(* IEC 61131-3 sources: std_i2980_v2.06_cp053/Source/IMM/ieccontrol/ODC1 (part 10) *)

@BEG_Export

@BEG_Algo
@POSTUPDATE_ALGORITHM @RT(21)pProgramSwitchChanged @STRUCTURED_TEXT
@RT(0) @RT(24)sv_bProgramSwitchChanged @RT(9)PU_Task_3 @F @F
@END_Algo

@BEG_Dcl
@RT(16)DclTreeContainer
0
@END_Dcl

@END_Export

@BEG_Export

@BEG_Algo
@POSTUPDATE_ALGORITHM @RT(18)pActivationChanged @STRUCTURED_TEXT
@RT(0) @RT(21)sv_bActivationChanged @RT(9)PU_Task_3 @F @F
@END_Algo

@BEG_Dcl
@RT(16)DclTreeContainer
0
@END_Dcl

@END_Export

@BEG_Export

@BEG_Algo
@PROCESS_ALGORITHM @RT(13)paVersionInfo @STRUCTURED_TEXT
@RT(0) @RT(0) @RT(8)TaskSlow @T @F
@END_Algo

@BEG_Dcl
@RT(16)DclTreeContainer
1
@Var @RT(1)b @RT(0) @T @F @DT @RT(4)BOOL @RT(0) @T @T @BASIC 0 @F
@F @F
@T
@BEG_Attrib
3 @RT(0) @RT(0) @RT(0)
@END_Attrib
1 0 @F @F @F @F

@END_Dcl

@END_Export

@BEG_Export

@BEG_Algo
@POSTUPDATE_ALGORITHM @RT(24)pChangeToProgramSwitches @STRUCTURED_TEXT
@RT(0) @RT(22)sv_bUseProgramSwitches @RT(9)PU_Task_7 @F @F
@END_Algo

@BEG_Dcl
@RT(16)DclTreeContainer
1
@Var @RT(7)iDevice @RT(0) @T @F @DT @RT(4)DINT @RT(0) @T @T @BASIC 0 @F
@F @F
@T
@BEG_Attrib
3 @RT(0) @RT(0) @RT(0)
@END_Attrib
1 4 @F @F @F @F

@END_Dcl

@END_Export

@BEG_Export

@BEG_Algo
@ALGORITHM @RT(26)aCheckCycleStartConditions @STRUCTURED_TEXT
@RT(0) @RT(0) @RT(0) @F @F
@END_Algo

@BEG_Dcl
@RT(16)DclTreeContainer
10
@Var @RT(3)Pos @RT(0) @T @T @DERIVED 0 @T @T @DT @RT(12)tsODCStepPos @RT(0) @T @T @UNKNOWN 0 @F
@F @F
@T
@BEG_Attrib
3 @RT(0) @RT(0) @RT(0)
@END_Attrib
1 0 @F @F @F @F

@Var @RT(8)DeviceId @RT(0) @T @T @DERIVED 0 @T @T @DT @RT(10)tsDeviceId @RT(0) @T @T @UNKNOWN 0 @F
@F @F
@T
@BEG_Attrib
3 @RT(0) @RT(0) @RT(0)
@END_Attrib
1 0 @F @F @F @F

@Var @RT(11)SafetyArray @RT(0) @T @T @DERIVED 0 @T @T @DT @RT(20)tyODCDependencyArray @RT(0) @T @T @UNKNOWN 0 @F
@F @F
@T
@BEG_Attrib
3 @RT(0) @RT(0) @RT(0)
@END_Attrib
1 0 @F @F @F @F

@Var @RT(12)iDefaultMove @RT(0) @T @F @DT @RT(4)DINT @RT(0) @T @T @BASIC 0 @F
@F @F
@T
@BEG_Attrib
3 @RT(0) @RT(0) @RT(0)
@END_Attrib
1 0 @F @F @F @F

@Var @RT(7)iDevice @RT(0) @T @F @DT @RT(4)DINT @RT(0) @T @T @BASIC 0 @F
@F @F
@T
@BEG_Attrib
3 @RT(0) @RT(0) @RT(0)
@END_Attrib
1 4 @F @F @F @F

@Var @RT(8)bAllowed @RT(0) @T @F @DT @RT(4)BOOL @RT(0) @T @T @BASIC 0 @F
@F @F
@T
@BEG_Attrib
3 @RT(0) @RT(0) @RT(0)
@END_Attrib
1 0 @F @F @F @F

@Var @RT(22)abODCCheckDependencies @RT(0) @T @T @DERIVED 0 @T @T @DT @RT(22)ABODCCheckDependencies @RT(0) @T @T @UNKNOWN 0 @F
@F @F
@T
@BEG_Attrib
3 @RT(0) @RT(0) @RT(0)
@END_Attrib
1 0 @F @F @F @F

@Var @RT(17)fbCheckPosReached @RT(0) @T @T @DERIVED 0 @T @T @DT @RT(17)FBCheckPosReached @RT(0) @T @T @UNKNOWN 0 @F
@F @F
@T
@BEG_Attrib
3 @RT(0) @RT(0) @RT(0)
@END_Attrib
1 0 @F @F @F @F

@Var @RT(15)bEjectorIgnored @RT(0) @T @F @DT @RT(4)BOOL @RT(0) @T @T @BASIC 0 @F
@F @F
@T
@BEG_Attrib
3 @RT(0) @RT(0) @RT(0)
@END_Attrib
1 0 @F @F @F @F

@Var @RT(17)EjectorDependency @RT(0) @T @F @DT @RT(5)LWORD @RT(0) @T @T @BASIC 0 @F
@F @F
@T
@BEG_Attrib
3 @RT(0) @RT(0) @RT(0)
@END_Attrib
1 0 @F @F @F @F

@END_Dcl

@END_Export

@BEG_Export

@BEG_Algo
@POSTUPDATE_ALGORITHM @RT(14)pOperationMode @STRUCTURED_TEXT
@RT(0) @RT(16)sv_OperationMode @RT(9)PU_Task_7 @F @F
@END_Algo

@BEG_Dcl
@RT(16)DclTreeContainer
2
@Var @RT(10)PrevOpMode @RT(0) @T @T @DERIVED 0 @T @T @DT @RT(15)tnOperationMode @RT(0) @T @T @UNKNOWN 0 @F
@F @F
@T
@BEG_Attrib
3 @RT(7)nManual @RT(0) @RT(0)
@END_Attrib
1 0 @F @F @F @F

@Var @RT(14)sOperationMode @RT(0) @T @F @DT @RT(11)STRING(255) @RT(0) @T @T @STRING 0 @F @RT(3)255 @F
@F @F
@T
@BEG_Attrib
3 @RT(0) @RT(0) @RT(0)
@END_Attrib
1 4 @F @F @F @F

@END_Dcl

@END_Export

@BEG_Export

@BEG_Algo
@PROCESS_ALGORITHM @RT(27)paRunManualCombinedMovement @SEQUENTIAL_FLOW_CHART
@RT(0) @RT(0) @RT(13)TaskSequencer @F @F
@END_Algo

@BEG_Dcl
@RT(16)DclTreeContainer
0
@END_Dcl

@END_Export

@BEG_Export

@BEG_Algo
@PROCESS_ALGORITHM @RT(23)paCheckConditionsManual @STRUCTURED_TEXT
@RT(0) @RT(0) @RT(10)TaskAnalog @F @F
@END_Algo

@BEG_Dcl
@RT(16)DclTreeContainer
2
@Var @RT(10)TmpStepPos @RT(0) @T @T @DERIVED 0 @T @T @DT @RT(12)tsODCStepPos @RT(0) @T @T @UNKNOWN 0 @F
@F @F
@T
@BEG_Attrib
3 @RT(0) @RT(0) @RT(0)
@END_Attrib
1 0 @F @F @F @F

@Var @RT(1)i @RT(0) @T @F @DT @RT(4)DINT @RT(0) @T @T @BASIC 0 @F
@F @F
@T
@BEG_Attrib
3 @RT(0) @RT(0) @RT(0)
@END_Attrib
1 4 @F @F @F @F

@END_Dcl

@END_Export

@BEG_Export

@BEG_Algo
@PROCESS_ALGORITHM @RT(11)paCycleTime @STRUCTURED_TEXT
@RT(0) @RT(0) @RT(10)TaskInject @F @F
@END_Algo

@BEG_Dcl
@RT(16)DclTreeContainer
2
@Var @RT(1)b @RT(0) @T @F @DT @RT(4)BOOL @RT(0) @T @T @BASIC 0 @F
@F @F
@T
@BEG_Attrib
3 @RT(0) @RT(0) @RT(0)
@END_Attrib
1 0 @F @F @F @F

@Var @RT(14)fbTonCycleTime @RT(0) @T @T @DERIVED 0 @T @T @DT @RT(3)TON @RT(0) @T @T @UNKNOWN 0 @F
@F @F
@T
@BEG_Attrib
3 @RT(0) @RT(0) @RT(0)
@END_Attrib
1 0 @F @F @F @F

@END_Dcl

@END_Export

@BEG_Export

@BEG_Algo
@PROCESS_ALGORITHM @RT(18)paCycleTimeMachine @STRUCTURED_TEXT
@RT(0) @RT(0) @RT(7)TaskMid @F @F
@END_Algo

@BEG_Dcl
@RT(16)DclTreeContainer
2
@Var @RT(1)b @RT(0) @T @F @DT @RT(4)BOOL @RT(0) @T @T @BASIC 0 @F
@F @F
@T
@BEG_Attrib
3 @RT(0) @RT(0) @RT(0)
@END_Attrib
1 0 @F @F @F @F

@Var @RT(21)fbTonCycleTimeMachine @RT(0) @T @T @DERIVED 0 @T @T @DT @RT(3)TON @RT(0) @T @T @UNKNOWN 0 @F
@F @F
@T
@BEG_Attrib
3 @RT(0) @RT(46)Clock the cycletime from start to end of cycle @RT(0)
@END_Attrib
1 0 @F @F @F @F

@END_Dcl

@END_Export

@BEG_Export

@BEG_Algo
@POSTUPDATE_ALGORITHM @RT(21)pSequenceInterruption @STRUCTURED_TEXT
@RT(0) @RT(24)sv_bSequenceInterruption @RT(10)PU_Task_13 @F @F
@END_Algo

@BEG_Dcl
@RT(16)DclTreeContainer
1
@Var @RT(5)dummy @RT(0) @T @F @DT @RT(4)DINT @RT(0) @T @T @BASIC 0 @F
@F @F
@T
@BEG_Attrib
3 @RT(0) @RT(0) @RT(0)
@END_Attrib
1 0 @F @F @F @F

@END_Dcl

@END_Export

@BEG_Export

@BEG_Algo
@ALGORITHM @RT(21)aStartInverseMovement @STRUCTURED_TEXT
@RT(0) @RT(0) @RT(0) @F @F
@END_Algo

@BEG_Dcl
@RT(16)DclTreeContainer
5
@Var @RT(7)iMoveNr @RT(0) @T @F @DT @RT(4)DINT @RT(0) @T @T @BASIC 0 @F
@F @F
@T
@BEG_Attrib
3 @RT(0) @RT(0) @RT(0)
@END_Attrib
1 1 @F @F @F @F

@Var @RT(7)iColumn @RT(0) @T @F @DT @RT(4)DINT @RT(0) @T @T @BASIC 0 @F
@F @F
@T
@BEG_Attrib
3 @RT(0) @RT(0) @RT(0)
@END_Attrib
1 1 @F @F @F @F

@Var @RT(8)iFuIndex @RT(0) @T @F @DT @RT(4)DINT @RT(0) @T @T @BASIC 0 @F
@F @F
@T
@BEG_Attrib
3 @RT(0) @RT(0) @RT(0)
@END_Attrib
1 0 @F @F @F @F

@Var @RT(14)iMoveIdInverse @RT(0) @T @T @DERIVED 0 @T @T @DT @RT(10)tMoveIdent @RT(0) @T @T @UNKNOWN 0 @F
@F @F
@T
@BEG_Attrib
3 @RT(0) @RT(0) @RT(0)
@END_Attrib
1 0 @F @F @F @F

@Var @RT(1)i @RT(0) @T @F @DT @RT(4)DINT @RT(0) @T @T @BASIC 0 @F
@F @F
@T
@BEG_Attrib
3 @RT(0) @RT(0) @RT(0)
@END_Attrib
1 4 @F @F @F @F

@END_Dcl

@END_Export

@BEG_Export

@BEG_Algo
@POSTUPDATE_ALGORITHM @RT(8)pStepFwd @STRUCTURED_TEXT
@RT(0) @RT(10)di_StepFwd @RT(9)PU_Task_3 @F @F
@END_Algo

@BEG_Dcl
@RT(16)DclTreeContainer
0
@END_Dcl

@END_Export

@BEG_Export

@BEG_Algo
@POSTUPDATE_ALGORITHM @RT(8)pStepBwd @STRUCTURED_TEXT
@RT(0) @RT(10)di_StepBwd @RT(9)PU_Task_3 @F @F
@END_Algo

@BEG_Dcl
@RT(16)DclTreeContainer
2
@Var @RT(7)iColumn @RT(0) @T @F @DT @RT(4)DINT @RT(0) @T @T @BASIC 0 @F
@F @F
@T
@BEG_Attrib
3 @RT(0) @RT(0) @RT(0)
@END_Attrib
1 4 @F @F @F @F

@Var @RT(13)iActiveMoveNr @RT(0) @T @F @DT @RT(4)DINT @RT(0) @T @T @BASIC 0 @F
@F @F
@T
@BEG_Attrib
3 @RT(0) @RT(0) @RT(0)
@END_Attrib
1 0 @F @F @F @F

@END_Dcl

@END_Export

@BEG_Export

@BEG_Algo
@EVENT_ALGORITHM @RT(28)evaModifyCycleStartCondition @STRUCTURED_TEXT
@RT(0) @RT(27)evModifyCycleStartCondition @RT(9)EV_Task_3 @F @F
@END_Algo

@BEG_Dcl
@RT(16)DclTreeContainer
8
@Var @RT(26)evModifyCycleStartCondData @RT(0) @T @T @DERIVED 0 @T @T @DT @RT(27)tevModifyCycleStartCondData @RT(0) @T @T @UNKNOWN 0 @F
@F @F
@T
@BEG_Attrib
3 @RT(0) @RT(0) @RT(0)
@END_Attrib
1 1 @F @F @F @F

@Var @RT(5)dummy @RT(0) @T @F @DT @RT(4)DINT @RT(0) @T @T @BASIC 0 @F
@F @F
@T
@BEG_Attrib
3 @RT(0) @RT(0) @RT(0)
@END_Attrib
1 0 @F @F @F @F

@Var @RT(9)eventData @RT(0) @T @T @DERIVED 0 @T @T @DT @RT(27)tevModifyCycleStartCondData @RT(0) @T @T @UNKNOWN 0 @F
@F @F
@T
@BEG_Attrib
3 @RT(0) @RT(0) @RT(0)
@END_Attrib
1 0 @F @F @F @F

@Var @RT(8)iFuIndex @RT(0) @T @F @DT @RT(4)DINT @RT(0) @T @T @BASIC 0 @F
@F @F
@T
@BEG_Attrib
3 @RT(0) @RT(0) @RT(0)
@END_Attrib
1 0 @F @F @F @F

@Var @RT(1)i @RT(0) @T @F @DT @RT(4)DINT @RT(0) @T @T @BASIC 0 @F
@F @F
@T
@BEG_Attrib
3 @RT(0) @RT(0) @RT(0)
@END_Attrib
1 4 @F @F @F @F

@Var @RT(7)iMoveNr @RT(0) @T @F @DT @RT(4)DINT @RT(0) @T @T @BASIC 0 @F
@F @F
@T
@BEG_Attrib
3 @RT(0) @RT(0) @RT(0)
@END_Attrib
1 0 @F @F @F @F

@Var @RT(15)fbAddDependency @RT(0) @T @T @DERIVED 0 @T @T @DT @RT(15)FBAddDependency @RT(0) @T @T @UNKNOWN 0 @F
@F @F
@T
@BEG_Attrib
3 @RT(0) @RT(0) @RT(0)
@END_Attrib
1 0 @F @F @F @F

@Var @RT(15)fbGetMoveNumber @RT(0) @T @T @DERIVED 0 @T @T @DT @RT(15)FBGetMoveNumber @RT(0) @T @T @UNKNOWN 0 @F
@F @F
@T
@BEG_Attrib
3 @RT(0) @RT(0) @RT(0)
@END_Attrib
1 0 @F @F @F @F

@END_Dcl

@END_Export

@BEG_Body
@TL(14)
(**************************************** WARNING ********************************************
 *** The KEBA Kemro K2 System including software is not intended for safety control tasks! ***
 ***                       For further information see Comment tab!                        ***
 *********************************************************************************************)

bActive := FALSE;
FOR i := 2 TO sv_iUsedColumns DO
   IF sv_InterpreterParallelInfo[i].bColumnActive THEN
      bActive := TRUE;
      EXIT;
   END_IF;
END_FOR;

@END_Body

@@@BEG_Comment@@@
@TL(0)

@@@END_Comment@@@

@BEG_Body
@TL(25)
(**************************************** WARNING ********************************************
 *** The KEBA Kemro K2 System including software is not intended for safety control tasks! ***
 ***                       For further information see Comment tab!                        ***
 *********************************************************************************************)

CycleTimeArray[i] := sv_dCycleTime;
dSum := dSum + CycleTimeArray[i];
i := i + 1;

IF i > cCycleTimeArraySize THEN
   //check if cycletime of last x - cycles is stable
   dAverageCycleTime := dSum / cCycleTimeArraySize;

   //-> check deviation between average cycle time and calculated cycle time
   IF (SUB_TIME(dAverageCycleTime, sv_dCalculatedCycleTime)) > sv_dAllowedCycleDeviation THEN
      sv_iEditorPropertiesChanged := sv_iEditorPropertiesChanged + 1;
   END_IF;

   i := 1;
   dSum := t#0s;
END_IF;

@END_Body

@@@BEG_Comment@@@
@TL(0)

@@@END_Comment@@@

@BEG_Body
@TL(34)
(**************************************** WARNING ********************************************
 *** The KEBA Kemro K2 System including software is not intended for safety control tasks! ***
 ***                       For further information see Comment tab!                        ***
 *********************************************************************************************)

IF NOT mbSequenceChanged THEN
   fbDebugTrace2(nODCInterpreter, 'no sequence backup written as sequence did NOT change');
   STOP_PROCESS_ALGORITHM();
   RETURN;
END_IF;

mbSequenceChanged := FALSE;

IF sv_ODCSequenceBackup[sv_iODCSequenceAct].Sequence = sv_ODCSequence THEN
   fbDebugTrace2(nODCInterpreter, 'ODC sequences equal, doing nothing');
   STOP_PROCESS_ALGORITHM();
   RETURN;
END_IF;
fbDebugTrace2(nODCInterpreter, 'ODC sequences different, making backup');

sv_iODCSequenceAct := sv_iODCSequenceAct + 1;
IF sv_iODCSequenceAct > cODCSequenceBackupCount THEN
   sv_iODCSequenceAct := 1;
END_IF;

//FIXME: maybe do in smaller steps to avoid blocking the system for a long time
fbDebugTrace2(nODCInterpreter, CONCAT('saving new ODC sequence in history at pos ', DINT_TO_STRING(sv_iODCSequenceAct)));

sv_ODCSequenceBackup[sv_iODCSequenceAct].Sequence := sv_ODCSequence;
sv_ODCSequenceBackup[sv_iODCSequenceAct].Date := sv_ODCSequenceGenerateTime;
fbDebugTrace2(nODCInterpreter, 'saving backup done');

STOP_PROCESS_ALGORITHM();

@END_Body

@@@BEG_Comment@@@
@TL(2)
Back up the current sequence (sv_ODCSequence)
A backup is only written when sv_ODCSequence is not equal to the last backup
@@@END_Comment@@@

@BEG_Body
@TL(10)
(**************************************** WARNING ********************************************
 *** The KEBA Kemro K2 System including software is not intended for safety control tasks! ***
 ***                       For further information see Comment tab!                        ***
 *********************************************************************************************)

IF RecalcMode > mPendingRecalc THEN
   mPendingRecalc := RecalcMode;
   sv_bRecalcPendingOrActive := TRUE;
END_IF;

@END_Body

@@@BEG_Comment@@@
@TL(5)
Queue a recalculation of the ODC sequence

nODCRecalcReloadFiles reload the ODC files from the CF + nODCRecalcCylce
nODCRecalcCylce       recalculate the cycle(because a program switch changed) + nODCRecalcSafety
nODCRecalcSafety      recalculate safety only(a movement was disabled)
@@@END_Comment@@@

@BEG_Body
@TL(44)
(**************************************** WARNING ********************************************
 *** The KEBA Kemro K2 System including software is not intended for safety control tasks! ***
 ***                       For further information see Comment tab!                        ***
 *********************************************************************************************)

bStartedRecalc := FALSE;

IF mPendingRecalc = nODCRecalcNone THEN
   RETURN;
END_IF;

IF mbRecalcActive THEN
   fbDebugTrace('another ODC recalc is already active, new recalc will be executed later');
   RETURN;
END_IF;

IF mPendingRecalc > mRecalcMode THEN
   mRecalcMode := mPendingRecalc;
END_IF;
// mRecalcMode will be reset after the recalc finished successfully
// but keeps the value if an error occured
// this way we can be sure the right recalc mode is used when
// the first recalc with nODCRecalcCylce fails and the second recalc with only nODCRecalcSafety succeeds
// the cycle is recalculated, and not only safety

mPendingRecalc := nODCRecalcNone;

IF mRecalcMode = nODCRecalcReloadFiles THEN
   fbDebugTrace2(nODCInterpreter, 'start initializing ODC array WITH reading new files');
ELSIF mRecalcMode = nODCRecalcCylce THEN
   fbDebugTrace2(nODCInterpreter, 'start initializing ODC array WITHOUT reading new files');
ELSIF mRecalcMode = nODCRecalcSafety THEN
   fbDebugTrace2(nODCInterpreter, 'start initializing ODC dependency array');
ELSIF mRecalcMode = nODCRecalcInternal THEN
   fbDebugTrace2(nODCInterpreter, 'start initializing internal ODC array');
ELSE
   fbDebugTrace2(nODCInterpreter, 'NOT starting initialization of ODC because we got a strange reason');
   RETURN;
END_IF;

bStartedRecalc := TRUE;
mbRecalcActive := TRUE; //set flag immediately, do not wait for PA, which might be delayed a bit because it is low prio
START_PROCESS_ALGORITHM(paInitSequence);

@END_Body

@@@BEG_Comment@@@
@TL(5)
Start a pending recalculation of the ODC sequence

If bStartedRecalc is TRUE then a pending recalculation was started.

To find out when recalculation finishes wait until mbRecalcActive is FALSE again
@@@END_Comment@@@

@BEG_SfcBody
60 37 52

@BEG_SfcData 2
@StepSeq @RT(4)sseq @F 15
@Step @RT(6)SError @F @F @T @F @RT(0) @F
@AcbCont @RT(7)unnamed @F 1
@Acb @RT(6)AError @F @T @RT(1)N @RT(0) @F @F @T @TL(22)
fbDebugTrace('initializing ODC array NOT successful');

(* set the generic erODCInitFailed ALARM which will block machine operation
   for detailed information other alarms are set which explain 1 or more problems
   of the ODC sequence *)
SET_ALARM(Name := erODCInitFailed);

mbRecalcActive := FALSE;

//reset mRecalcMode
//this way a failed recalc can not be replaced by a succeeding recalc
//of lower priority
mRecalcMode := FailedRecalc;

// indicate an update of the odc list so the hmi can react properly
sv_iODCSequenceUpdated := sv_iODCSequenceUpdated + 1;

//notify other code parts when recalc is finished (in this case unsuccessfully)
sv_bRecalcPendingOrActive := FALSE;

STOP_PROCESS_ALGORITHM();

@F

@Trans @RT(7)Trans25 @F @T @F @F @T @T @TL(2)
TRUE

@RT(7)Trans25 @F
@Step @RT(6)SStart @F @T @T @F @RT(0) @F
@AcbCont @RT(7)unnamed @F 3
@Acb @RT(6)AStart @F @T @RT(1)P @RT(0) @F @F @T @TL(14)
fbDebugTrace2(nODCInterpreter, 'starting initialisation of ODC sequence');

RESET_ALARM(Name := erODCInitFailed);

RecalcMode := mRecalcMode;
FailedRecalc := mRecalcMode;  //remember in case of failed recalc so we can repeat
mRecalcMode := nODCRecalcNone;

sv_iInitOK := 0;

(* lock all movements so nothing can happen during init *)
fbLockUnlockAll.Alarm.AlarmId := erMachineSequenceNotCreated;
fbLockUnlockAll(Mode := nLockAbort);

@F
@Acb @RT(23)AInitAdditionalMoveData @F @F @RT(1)P @RT(0) @F @F @F @F
@Acb @RT(26)AResetProgrammedInSequence @F @F @RT(1)P @RT(0) @F @F @F @F

@AltBranch @RT(3)alt @F 2
@TransSeq @RT(4)tseq @F 1
@Trans @RT(7)Trans38 @F @T @F @F @T @F @TL(2)
RecalcMode <> nODCRecalcInternal

@RT(7)Trans38 @F

@TransSeq @RT(4)tseq @F 2
@Trans @RT(22)TNewSequenceFromEditor @F @T @F @F @T @F @TL(2)
RecalcMode = nODCRecalcInternal

@RT(7)Trans39 @F
@Goto @RT(21)SSanityCheckAndNumber @F @F

@Step @RT(6)Step28 @F @F @F @F @RT(0) @F
@AcbCont @RT(7)unnamed @F 0

@AltBranch @RT(3)alt @F 2
@TransSeq @RT(4)tseq @F 1
@Trans @RT(7)Trans13 @F @T @F @F @T @F @TL(2)
NOT (RecalcMode >= nODCRecalcReloadFiles)

@RT(7)Trans13 @F

@TransSeq @RT(4)tseq @F 5
@Trans @RT(18)TRecalcReloadFiles @F @T @F @F @T @F @TL(2)
RecalcMode >= nODCRecalcReloadFiles

@RT(7)Trans12 @F
@Step @RT(13)SInitSequence @F @F @F @F @RT(0) @F
@AcbCont @RT(7)unnamed @F 2
@Acb @RT(6)AInit1 @F @T @RT(1)P @RT(0) @F @F @T @TL(11)
iCalledInit := 0;
iCalledCreate := 0;

IF NOT bFirstCall THEN
   sWorkPath := FGetCatConfigValueString('System.workPath', '/harddisk0/');
   bFirstCall := TRUE;
END_IF;

sPath := CONCAT(sWorkPath, sv_ODCDescriptionPath);
abKODC_Builder.Init(Movements := sv_ODCMovements, DescriptionFilePath := sPath, Execute := FALSE);

@F
@Acb @RT(6)AInit2 @F @T @RT(1)N @RT(0) @F @F @T @TL(3)
abKODC_Builder.Init(Execute := TRUE);
iCalledInit := iCalledInit + 1;

@F

@Trans @RT(6)Trans2 @F @T @F @F @T @T @TL(2)
abKODC_Builder.Init.Done OR abKODC_Builder.Init.Error

@RT(6)Trans2 @F
@Step @RT(17)SInitSequenceDone @F @F @F @F @RT(0) @F
@AcbCont @RT(7)unnamed @F 1
@Acb @RT(6)AInit3 @F @T @RT(1)P @RT(0) @F @F @T @TL(14)
IF abKODC_Builder.Init.Error AND abKODC_Builder.Init.Done THEN
   fbDebugTrace2(nODCInterpreter, 'ERROR init returned success and failure at the same time');
END_IF;

IF abKODC_Builder.Init.Done THEN
   fbDebugTrace2(nODCInterpreter, CONCAT('called init ',
                                         DINT_TO_STRING(iCalledInit),
                                         ' times then it returned success'));
ELSIF abKODC_Builder.Init.Error THEN
   fbDebugTrace2(nODCInterpreter, CONCAT('called init ',
                                         DINT_TO_STRING(iCalledInit),
                                         ' times then it returned error'));
END_IF;

@F

@AltBranch @RT(3)alt @F 2
@TransSeq @RT(4)tseq @F 1
@Trans @RT(7)Trans11 @F @T @F @F @T @F @TL(2)
NOT abKODC_Builder.Init.Error

@RT(7)Trans11 @F

@TransSeq @RT(4)tseq @F 2
@Trans @RT(7)Trans26 @F @T @F @F @T @F @TL(2)
abKODC_Builder.Init.Error

@RT(7)Trans26 @F
@Goto @RT(6)SError @F @F

@Step @RT(6)Step16 @F @F @F @F @RT(0) @F
@AcbCont @RT(7)unnamed @F 0

@AltBranch @RT(3)alt @F 2
@TransSeq @RT(4)tseq @F 1
@Trans @RT(7)Trans20 @F @T @F @F @T @F @TL(2)
NOT (RecalcMode >= nODCRecalcCylce)

@RT(7)Trans20 @F

@TransSeq @RT(4)tseq @F 11
@Trans @RT(12)TRecalcCycle @F @T @F @F @T @F @TL(2)
RecalcMode >= nODCRecalcCylce

@RT(7)Trans19 @F
@Step @RT(15)SCreateSequence @F @F @F @F @RT(0) @F
@AcbCont @RT(7)unnamed @F 3
@Acb @RT(14)AClearSequence @F @F @RT(1)P @RT(0) @F @F @T @F
@Acb @RT(16)ACreateSequence1 @F @T @RT(1)P @RT(0) @F @F @T @TL(6)
fbDebugTrace2(nODCInterpreter, 'initialisation of ODC array');
(* WARNING: Columns and Rows must be <= the real size of the array
   otherwise the builder will write outside of the array
   and memory corruption will occur ! *)
abKODC_Builder.CreateSequence(Sequence := sv_ODCSequence, Columns := cMaxParallelMovements, Rows := cMaxODCSteps, Execute := FALSE);

@F
@Acb @RT(16)ACreateSequence2 @F @T @RT(1)N @RT(0) @F @F @T @TL(3)
abKODC_Builder.CreateSequence(Execute := TRUE);
iCalledCreate := iCalledCreate + 1;

@F

@Trans @RT(6)Trans4 @F @T @F @F @T @T @TL(2)
abKODC_Builder.CreateSequence.Error OR abKODC_Builder.CreateSequence.Done

@RT(6)Trans4 @F
@Step @RT(19)SCreateSequenceDone @F @F @F @F @RT(0) @F
@AcbCont @RT(7)unnamed @F 1
@Acb @RT(16)ACreateSequence3 @F @T @RT(1)P @RT(0) @F @F @T @TL(14)
IF abKODC_Builder.CreateSequence.Error AND abKODC_Builder.CreateSequence.Done THEN
   fbDebugTrace2(nODCInterpreter, 'ERROR CreateSequence returned success and failure at the same time');
END_IF;

IF abKODC_Builder.CreateSequence.Done THEN
   fbDebugTrace2(nODCInterpreter, CONCAT('called CreateSequence ',
                                         DINT_TO_STRING(iCalledCreate),
                                         ' times then it returned success'));
ELSIF abKODC_Builder.CreateSequence.Error THEN
   fbDebugTrace2(nODCInterpreter, CONCAT('called CreateSequence ',
                                         DINT_TO_STRING(iCalledCreate),
                                         ' times then it returned error'));
END_IF;

@F

@AltBranch @RT(3)alt @F 2
@TransSeq @RT(4)tseq @F 1
@Trans @RT(7)Trans27 @F @T @F @F @T @F @TL(2)
NOT abKODC_Builder.CreateSequence.Error

@RT(7)Trans27 @F

@TransSeq @RT(4)tseq @F 2
@Trans @RT(7)Trans28 @F @T @F @F @T @F @TL(2)
abKODC_Builder.CreateSequence.Error

@RT(7)Trans28 @F
@Goto @RT(6)SError @F @F

@Step @RT(21)SSanityCheckAndNumber @F @F @T @F @RT(0) @F
@AcbCont @RT(7)unnamed @F 3
@Acb @RT(23)ACheckSequenceDimension @F @F @RT(1)P @RT(0) @F @F @F @F
@Acb @RT(15)AInitEmptySteps @F @F @RT(1)P @RT(0) @F @F @F @F
@Acb @RT(7)ASanity @F @T @RT(1)P @RT(0) @F @F @T @TL(10)
bError := FALSE;
abInterpreter.aCheckSequenceSanity();
IF NOT abInterpreter.aCheckSequenceSanity.bOK THEN
   fbDebugTrace('checking sanity of ODC array failed');
   bError := TRUE;
   RETURN;
END_IF;
bAddLoop := NOT abInterpreter.aCheckSequenceSanity.bAutoCycleLoopFound;
iNoOfStartParallel := abInterpreter.aCheckSequenceSanity.iNoOfStartParallel;

@F

@AltBranch @RT(3)alt @F 2
@TransSeq @RT(4)tseq @F 1
@Trans @RT(7)Trans46 @F @T @F @F @T @F @TL(2)
NOT bError

@RT(7)Trans46 @F

@TransSeq @RT(4)tseq @F 2
@Trans @RT(7)Trans50 @F @T @F @F @T @F @TL(2)
bError

@RT(7)Trans50 @F
@Goto @RT(6)SError @F @F

@Step @RT(6)Step33 @F @F @F @F @RT(0) @F
@AcbCont @RT(7)unnamed @F 0

@AltBranch @RT(3)alt @F 2
@TransSeq @RT(4)tseq @F 3
@Trans @RT(7)Trans48 @F @T @F @F @T @F @TL(2)
bAddLoop

@RT(7)Trans48 @F
@Step @RT(14)S_AddCycleLoop @F @F @F @F @RT(0) @F
@AcbCont @RT(7)unnamed @F 1
@Acb @RT(20)AInsertAutoCycleLoop @F @F @RT(1)P @RT(0) @F @F @F @F

@Trans @RT(10)TLoopAdded @F @T @F @F @T @T @TL(2)
TRUE

@RT(7)Trans50 @F

@TransSeq @RT(4)tseq @F 1
@Trans @RT(7)Trans49 @F @T @T @F @T @F @TL(2)
NOT bAddLoop

@RT(7)Trans49 @F

@Step @RT(6)Step32 @F @F @F @F @RT(0) @F
@AcbCont @RT(7)unnamed @F 1
@Acb @RT(23)ACreateInternalSequence @F @T @RT(1)P @RT(0) @F @F @T @TL(18)
bError := FALSE;
abInterpreter.aClearInternalSequence();

abInterpreter.aCreateInternalSequence();
IF abInterpreter.aCreateInternalSequence.bError THEN
   fbDebugTrace('aCreateInternalSequence failed');
   bError := TRUE;
   RETURN;
END_IF;

sv_iUsedColumns := abInterpreter.aCreateInternalSequence.iUsedColumns;
sv_iUsedRows := abInterpreter.aCreateInternalSequence.iUsedRows;

// save sequence generation time
fbRTC(EN := FALSE);
sv_ODCSequenceGenerateTime := fbRTC.CDT;
mbSequenceChanged := TRUE;

@F

@AltBranch @RT(3)alt @F 2
@TransSeq @RT(4)tseq @F 3
@Trans @RT(7)Trans14 @F @T @F @F @T @T @TL(2)
NOT bError

@RT(7)Trans14 @F
@Step @RT(6)Step26 @F @F @F @F @RT(0) @F
@AcbCont @RT(7)unnamed @F 1
@Acb @RT(15)AInitSequenceOK @F @T @RT(1)N @RT(0) @F @F @T @TL(2)
sv_iInitOK := 10;

@F

@Trans @RT(7)Trans36 @F @T @F @F @T @F @TL(2)
TRUE

@RT(7)Trans36 @F

@TransSeq @RT(4)tseq @F 2
@Trans @RT(7)Trans29 @F @T @F @F @T @T @TL(2)
bError

@RT(7)Trans29 @F
@Goto @RT(6)SError @F @F

@Step @RT(19)SBeforeRecalcSafety @F @F @F @F @RT(0) @F
@AcbCont @RT(7)unnamed @F 0

@AltBranch @RT(3)alt @F 2
@TransSeq @RT(4)tseq @F 1
@Trans @RT(7)Trans22 @F @T @F @F @T @F @TL(2)
NOT (RecalcMode >= nODCRecalcSafety)

@RT(7)Trans22 @F

@TransSeq @RT(4)tseq @F 3
@Trans @RT(13)TRecalcSafety @F @T @F @F @T @F @TL(2)
RecalcMode >= nODCRecalcSafety

@RT(7)Trans23 @F
@Step @RT(13)SRecalcSafety @F @F @F @F @RT(0) @F
@AcbCont @RT(7)unnamed @F 2
@Acb @RT(20)ACalcSeqDependencies @F @T @RT(1)P @RT(0) @F @F @T @TL(11)
IF iNoOfStartParallel <= cMaxStartParallel THEN
   RESET_ALARM(Name := erTooManyStartParallel);
   abSequDependencies.aCalc();
   IF abSequDependencies.aCalc.bError THEN
      bError := TRUE;
      fbDebugTrace('sequence dependency calculation returned a error');
   END_IF;
ELSE
   SET_ALARM(Name := erTooManyStartParallel);
END_IF;

@F
@Acb @RT(24)ASetProgrammedInSequence @F @F @RT(1)P @RT(0) @F @F @F @F

@AltBranch @RT(3)alt @F 2
@TransSeq @RT(4)tseq @F 1
@Trans @RT(7)Trans24 @F @T @F @F @T @F @TL(2)
NOT bError

@RT(7)Trans24 @F

@TransSeq @RT(4)tseq @F 2
@Trans @RT(7)Trans30 @F @T @F @F @T @F @TL(2)
bError

@RT(7)Trans30 @F
@Goto @RT(6)SError @F @F

@Step @RT(22)S_Check_Pending_Recalc @F @F @F @F @RT(0) @F
@AcbCont @RT(7)unnamed @F 1
@Acb @RT(22)ACheckForPendingRecalc @F @T @RT(1)P @RT(0) @F @F @T @TL(9)
bTryAgain := FALSE;
IF mPendingRecalc <> nODCRecalcNone THEN
   //recalc during creation of sequence requested
   //=> ignore result and start again
   mRecalcMode := mPendingRecalc;
   mPendingRecalc := nODCRecalcNone;
   bTryAgain := TRUE;
END_IF;

@F

@AltBranch @RT(3)alt @F 2
@TransSeq @RT(4)tseq @F 1
@Trans @RT(9)TNoRecalc @F @T @F @F @T @F @TL(2)
NOT bTryAgain

@RT(7)Trans44 @F

@TransSeq @RT(4)tseq @F 2
@Trans @RT(7)TRecalc @F @T @F @F @T @F @TL(2)
bTryAgain

@RT(7)Trans45 @F
@Goto @RT(6)SStart @F @F

@Step @RT(7)SFinish @F @F @F @F @RT(0) @F
@AcbCont @RT(7)unnamed @F 2
@Acb @RT(24)ACheckEjeBwdAtCycleStart @F @F @RT(1)P @RT(0) @F @F @F @F
@Acb @RT(7)AFinish @F @T @RT(1)N @RT(0) @F @F @T @TL(18)
(* array ok -> unlock all movements *)
fbLockUnlockAll.Alarm.AlarmId := erMachineSequenceNotCreated;
fbLockUnlockAll(Mode := nUnlock);

abInterpreter.aSetInitOK();
fbDebugTrace2(nODCInterpreter, 'initializing ODC array successful');

mbRecalcActive := FALSE;

// indicate an update of the odc list so the hmi can react properly
sv_iInitOK := 20;
sv_iODCSequenceUpdated := sv_iODCSequenceUpdated + 1;

//notify other code parts when recalc is finished (and it is OK to send an evStartRequest)
sv_bRecalcPendingOrActive := FALSE;

STOP_PROCESS_ALGORITHM();

@F

@Trans @RT(6)Trans8 @F @T @F @F @T @T @TL(2)
TRUE

@RT(6)Trans8 @F
@Goto @RT(6)SStart @F @F
@END_SfcData
@SaActions 8
@SaText @RT(14)AClearSequence 1 @TL(9)
(* make sure the array is clean
   important for testing when 2 different partially initialized
   arrays are used *)
FOR iTmpCol := 1 TO cMaxParallelMovements DO
   FOR iTmpRow := 1 TO cMaxODCSteps DO
      sv_ODCSequence[iTmpCol][iTmpRow] := EmptySequenceEntry;
   END_FOR;
END_FOR;

@SaText @RT(23)AInitAdditionalMoveData 1 @TL(35)
(**************************************** WARNING ********************************************
 *** The KEBA Kemro K2 System including software is not intended for safety control tasks! ***
 ***                       For further information see Comment tab!                        ***
 *********************************************************************************************)
IF NOT bInitDone THEN

   //get FuIndex of all registered movements
   //fuIndex = index of the device in sv_ODCDeviceMovements
   FOR iMove := 1 TO sv_iMovementsAvailable DO
      FOR iDevice := 1 TO sv_ODCDeviceMovements.iCount DO
         IF sv_MovementsAvailable[iMove].DeviceId = sv_ODCDeviceMovements.Devices[iDevice].DeviceId THEN
            sv_MovementsAvailable[iMove].iFuIndex := iDevice;
            EXIT;
         END_IF;
      END_FOR;
   END_FOR;

   //get number of default movement for every device in sv_ODCDeviceMovements
   FOR iDevice := 1 TO sv_ODCDeviceMovements.iCount DO
      DeviceId := sv_ODCDeviceMovements.Devices[iDevice].DeviceId;
      FOR iMove := 1 TO sv_iMovementsAvailable DO
         IF sv_MovementsAvailable[iMove].DeviceId = DeviceId AND sv_MovementsAvailable[iMove].pMovementData^.bDefaultPos THEN
            //default movement found
            sv_ODCDeviceMovements.Devices[iDevice].iDefaultMoveNumber := iMove;
            EXIT;
         END_IF;
      END_FOR;
   END_FOR;

   bInitDone := TRUE;

END_IF;

@SaText @RT(26)AResetProgrammedInSequence 1 @TL(33)
(**************************************** WARNING ********************************************
 *** The KEBA Kemro K2 System including software is not intended for safety control tasks! ***
 ***                       For further information see Comment tab!                        ***
 *********************************************************************************************)

IF RecalcMode = nODCRecalcNone OR RecalcMode = nODCRecalcSafety THEN
   ;//no change in sequence
ELSE
   //sequence changed -> reset bProgrammedInSequence for all movements
   FOR iMove := 1 TO sv_iMovementsAvailable DO
      sv_MovementsAvailable[iMove].pMovementData^.bProgrammedInSequence := FALSE;

      IF sv_MovementsAvailable[iMove].pMovementData^.bInstanceable AND
        CHECK_REF(sv_MovementsAvailable[iMove].pMovementData^.InstanceData.pProgrammedInSequenceArray^) THEN

         //movement instanceable -> init programmed in sequence for all instances
         FOR k:= 1 TO cMaxIntermediateConditions DO
            sv_MovementsAvailable[iMove].pMovementData^.InstanceData.pProgrammedInSequenceArray^[k] := FALSE;
         END_FOR;

      END_IF;
   END_FOR;

   //reset array with start condition positions
   FOR i := 1 TO cMaxStartConditions DO
      mStartConditionPosArray[i].iColumn := 0;
      mStartConditionPosArray[i].iRow := 0;
   END_FOR;
END_IF;

@SaText @RT(24)ASetProgrammedInSequence 1 @TL(32)
(**************************************** WARNING ********************************************
 *** The KEBA Kemro K2 System including software is not intended for safety control tasks! ***
 ***                       For further information see Comment tab!                        ***
 *********************************************************************************************)

//set bProgrammedInSequence for all movements which are
//included in the created sequence
FOR iTmpRow := 1 TO sv_iUsedRows DO
   FOR iTmpCol := 1 TO sv_iUsedColumns DO
      iMove := sv_ODCSequenceInt[iTmpCol,iTmpRow].iMoveNumber;
      IF iMove >= cMoveNone THEN
         sv_MovementsAvailable[iMove].pMovementData^.bProgrammedInSequence := TRUE;

         IF sv_MovementsAvailable[iMove].pMovementData^.bInstanceable AND
           CHECK_REF(sv_MovementsAvailable[iMove].pMovementData^.InstanceData.pProgrammedInSequenceArray^) THEN
            //movement instanceable -> set programmed in sequence for according instance
            iInstance := sv_ODCSequenceInt[iTmpCol,iTmpRow].iCount;
            sv_MovementsAvailable[iMove].pMovementData^.InstanceData.pProgrammedInSequenceArray^[iInstance] := TRUE;
         END_IF;

      END_IF;

      //save position if step is a start condition
      IF sv_ODCSequence[iTmpCol,iTmpRow].iMoveId = cMoveStartCondition THEN
         iCount := sv_ODCSequence[iTmpCol, iTmpRow].iCount;
         mStartConditionPosArray[iCount].iColumn := iTmpCol;
         mStartConditionPosArray[iCount].iRow := iTmpRow;
      END_IF;

   END_FOR;
END_FOR;

@SaText @RT(24)ACheckEjeBwdAtCycleStart 1 @TL(40)
(**************************************** WARNING ********************************************
 *** The KEBA Kemro K2 System including software is not intended for safety control tasks! ***
 ***                       For further information see Comment tab!                        ***
 *********************************************************************************************)

//get index of ejector 1 in sv_ODCDeviceMovements
//and also get dependency which represents "Ejector bwd"
IF NOT bInit THEN
   FOR i := 1 TO g_iODCMoveDevicesRegistered DO
      IF sv_ODCDeviceMovements.Devices[i].DeviceId = DeviceIdEjector1 THEN
         miIndexEjectorInSafetyArray := i;

         //find ejector bwd movement
         FOR k := 1 TO sv_ODCDeviceMovements.Devices[miIndexEjectorInSafetyArray].iNumberOfMovements DO
            IF sv_ODCDeviceMovements.Devices[miIndexEjectorInSafetyArray].Movements[k]^.MoveId = cMoveBwd THEN

               //movement found in sv_ODCDeviceMovements -> set the according bit
               DependencyEjectorBwd := cFirstBit;

               //first movement: shift right 0, second movement: shift right 1, ...
               DependencyEjectorBwd := SHR(DependencyEjectorBwd, (k-1));
               EXIT;
            END_IF;
         END_FOR;

         EXIT;
      END_IF;
   END_FOR;
   bInit := TRUE;
END_IF;

//avoid problems if no ejector is available
mbEjeBwdAtCycleStart := FALSE;
IF miIndexEjectorInSafetyArray > 0 THEN
   //check dependency array of first step and find out if ejector must be bwd
   IF sv_ODCSequenceInt[1,1].SafetyArray[miIndexEjectorInSafetyArray].Dependency = DependencyEjectorBwd THEN
      mbEjeBwdAtCycleStart := TRUE;
   END_IF;
END_IF;

@SaText @RT(20)AInsertAutoCycleLoop 1 @TL(50)
(**************************************** WARNING ********************************************
 *** The KEBA Kemro K2 System including software is not intended for safety control tasks! ***
 ***                       For further information see Comment tab!                        ***
 *********************************************************************************************)

IF sv_TraceLevel.bODCInterpreter THEN
   dummy := Print('No AutoCycleLoop found ----> add LOOP automatically');
END_IF;

iOrigEndLine := abInterpreter.aCheckSequenceSanity.iEndSequenceRow;
IF sv_TraceLevel.bODCInterpreter THEN
   dummy := Print('original end line: %d', iOrigEndLine);
END_IF;

//move line with ODC.EndSequence two lines down
//add ODC.EndLoop before ODC.EndSequence
//move the whole sequence one line down
//add ODC.BeginLoop in second line (first line is ODC.BeginSequence)
//fill sv_LoopData with correct values

FOR iTmpCol2 := 1 TO cMaxParallelMovements DO
   sv_ODCSequence[iTmpCol2,(iOrigEndLine+2)] := sv_ODCSequence[iTmpCol2, iOrigEndLine];
END_FOR;

IF sv_TraceLevel.bODCInterpreter THEN
   iTmp := iOrigEndLine +1;
   dummy := Print('Adding end loop in line %d', iTmp);
END_IF;

sv_ODCSequence[1,(iOrigEndLine+1)] := StepEndLoop;
g_iAutoCycleLoopEndLine := (iOrigEndLine+1);

FOR iTmpRow2 := iOrigEndLine TO 2 BY -1 DO
   FOR iTmpCol2 := 1 TO cMaxParallelMovements DO
      sv_ODCSequence[iTmpCol2,iTmpRow2] := sv_ODCSequence[iTmpCol2,(iTmpRow2-1)];
   END_FOR;
END_FOR;

IF sv_TraceLevel.bODCInterpreter THEN
   dummy := Print('Adding begin loop in line 2');
END_IF;
sv_ODCSequence[1,2] := StepBeginLoop;
g_iAutoCycleLoopStartLine := 2;

sv_LoopParameter[1].sTextKey := 'TxtAutoCycleLoop';
sv_LoopParameter[1].sVariable1 := 'system.sv_bFALSE';
sv_LoopParameter[1].sVariable2 := 'system.sv_bTRUE';
sv_LoopParameter[1].CompareOperator := nCompOperatorEqual;

@SaText @RT(15)AInitEmptySteps 1 @TL(18)
(**************************************** WARNING ********************************************
 *** The KEBA Kemro K2 System including software is not intended for safety control tasks! ***
 ***                       For further information see Comment tab!                        ***
 *********************************************************************************************)

//performance optimization:
//at empty steps the machine sequencer only sets iCompId to cMinCompId
//iMoveId, iMoveDir, ... are not changed and keep the "old" values
//=> this steps must be set to "empty" steps in the IEC code
FOR iTmpCol := 1 TO cMaxParallelMovements DO
   FOR iTmpRow := 1 TO cMaxODCSteps DO
      IF (sv_ODCSequence[iTmpCol][iTmpRow].iCompId = cMinCompId) AND (sv_ODCSequence[iTmpCol][iTmpRow].iMoveId <> cMoveNone) THEN
         //set the whole step to "Empty"
         sv_ODCSequence[iTmpCol][iTmpRow] := EmptySequenceEntry;
      END_IF;
   END_FOR;
END_FOR;

@SaText @RT(23)ACheckSequenceDimension 1 @TL(38)
(**************************************** WARNING ********************************************
 *** The KEBA Kemro K2 System including software is not intended for safety control tasks! ***
 ***                       For further information see Comment tab!                        ***
 *********************************************************************************************)

IF (sv_SequenceDimension.iMaxColumns > 0) AND (sv_SequenceDimension.iMaxRows > 0) THEN

   IF sv_SequenceDimension.iMaxColumns < cMaxParallelMovements THEN
      //loaded sequence is smaller (lower number of columns) than the actual sequence
      //-> init the rest of the columns
      FOR iTmpCol := (sv_SequenceDimension.iMaxColumns + 1) TO cMaxParallelMovements DO
         FOR iTmpRow := 1 TO cMaxODCSteps DO
            sv_ODCSequence[iTmpCol][iTmpRow] := EmptySequenceEntry;
         END_FOR;
      END_FOR;
   END_IF;

   IF sv_SequenceDimension.iMaxRows < cMaxODCSteps THEN
      //loaded sequence is smaller (lower number of rows) than the actual sequence
      //-> init the rest of the rows
      FOR iTmpCol := 1 TO sv_SequenceDimension.iMaxColumns DO
         FOR iTmpRow := (sv_SequenceDimension.iMaxRows + 1) TO cMaxODCSteps DO
            sv_ODCSequence[iTmpCol][iTmpRow] := EmptySequenceEntry;
         END_FOR;
      END_FOR;
   END_IF;
ELSE
   ;//loaded data does not contain the sequence dimension (=> data was created with a KePlast version < 01.38)
   //Attention:
   //It is not possible to automatically assume that the sequence dimension is 6 columns and 100 rows
   //in this case, because maybe in some customer projects the sequence size was already increased in
   //KePlast versions < 01.38
END_IF;

//set dimension to actual implemented array size
sv_SequenceDimension.iMaxColumns := cMaxParallelMovements;
sv_SequenceDimension.iMaxRows := cMaxODCSteps;

@SaTrans 0
@SaExits 0
@END_SfcBody

@@@BEG_Comment@@@
@TL(3)
Does the (re)initialisation of the ODC sequence and saves
the sequence generation time

@@@END_Comment@@@

@BEG_Body
@TL(24)
(**************************************** WARNING ********************************************
 *** The KEBA Kemro K2 System including software is not intended for safety control tasks! ***
 ***                       For further information see Comment tab!                        ***
 *********************************************************************************************)

fbDebugTrace2(nODCInterpreter, 'begin clearing step state');

FOR iTmpRow := 1 TO sv_iUsedRows DO
   fbSetStepState.StepState := nStateDefault;
   fbSetStepState.StepPos.iRow := iTmpRow;

   FOR iTmpColumn := 1 TO sv_iUsedColumns DO
      fbSetStepState.StepPos.iColumn := iTmpColumn;

      IF NOT (bExcludeActiveColumns AND sv_InterpreterParallelInfo[iTmpColumn].bColumnActive) THEN
         //reset step state depending on bExcludeActiceColumns
         fbSetStepState();
      END_IF;

   END_FOR;
END_FOR;

fbDebugTrace2(nODCInterpreter, 'finished clearing step state');

@END_Body

@@@BEG_Comment@@@
@TL(0)

@@@END_Comment@@@

@BEG_Body
@TL(64)
(**************************************** WARNING ********************************************
 *** The KEBA Kemro K2 System including software is not intended for safety control tasks! ***
 ***                       For further information see Comment tab!                        ***
 *********************************************************************************************)

// check if a start condition exists for the requested movement
bStartConditionOk := TRUE;
iStartConditionsNotOk := 0;
FOR i := 1 TO cMaxStartConditions DO
   IF sv_ODCSequence[StepPos.iColumn][StepPos.iRow] = sv_StartConditionInstanceData[i].DelayedMovement THEN
      // start condition found -> check if start condition is reached
      abInterpreter.aCheckStartConditionReached(iInstance := i);
      IF NOT abInterpreter.aCheckStartConditionReached.bReached THEN
         IF NOT bNoAlarms THEN
            // set alarm
            SET_ALARM(Name := erCompNotInCorrectPosition,
                      SubID1 := sv_StartConditionInstanceData[i].RelatedMovement.iCompId,
                      SubID2 := sv_StartConditionInstanceData[i].RelatedMovement.iIndexId);
         END_IF;
         bStartConditionOk := FALSE;
         iStartConditionsNotOk := iStartConditionsNotOk + 1;
      END_IF;
   ELSIF sv_ODCSequence[StepPos.iColumn][StepPos.iRow] = sv_StartConditionInstanceData[i].RelatedMovement THEN
      //also check if the requested movement is the "RelatedMovement" of a startcondition
      //for example: core in with startpos parallel to mold close
      //if mold close movement is requested, the core must be out until the start position for the core is reached

      //check if start condition is reached
      abInterpreter.aCheckStartConditionReached(iInstance := i);
      IF NOT abInterpreter.aCheckStartConditionReached.bReached THEN
         //check safety array
         abODCCheckDependencies.aCheck.StepPos.iColumn := mStartConditionPosArray[i].iColumn;
         abODCCheckDependencies.aCheck.StepPos.iRow := mStartConditionPosArray[i].iRow;

         abODCCheckDependencies.aCheck(DeviceIdSelf := sv_DeviceId, bNoAlarmsAndStepState := bNoAlarms);
         IF NOT abODCCheckDependencies.aCheck.bAllowed THEN
            fbDebugTrace2(nODCInterpreter, CONCAT('manual movement at pos ',
                                                   DINT_TO_STRING(StepPos.iRow),
                                                   '/',
                                                   DINT_TO_STRING(StepPos.iColumn),
                                                   ' not allowed because of related startcondition'));
            bStartConditionOk := FALSE;
            iStartConditionsNotOk := iStartConditionsNotOk + 1;
         END_IF;
      END_IF;
   END_IF;
END_FOR;

// check if a check condition exists for the requested movement
bCheckConditionsOk := TRUE;
bCheckConditionFound := FALSE;
iCheckConditionsNotOk := 0;
abInterpreter.aFindCheckCondition(Movement := sv_ODCSequence[StepPos.iColumn][StepPos.iRow],
                                    bFound => bCheckConditionFound);

IF bCheckConditionFound THEN
   abInterpreter.aCheckConditionsManual(Movement := sv_ODCSequence[StepPos.iColumn][StepPos.iRow], bNoAlarms := bNoAlarms);
   bCheckConditionsOk := abInterpreter.aCheckConditionsManual.bCheckConditionsOk;
   iCheckConditionsNotOk := abInterpreter.aCheckConditionsManual.iConditionsNotOk;
END_IF;

@END_Body

@@@BEG_Comment@@@
@TL(1)
Start a single movement (in response to evStartRequest)
@@@END_Comment@@@

@BEG_Body
@TL(149)
(**************************************** WARNING ********************************************
 *** The KEBA Kemro K2 System including software is not intended for safety control tasks! ***
 ***                       For further information see Comment tab!                        ***
 *********************************************************************************************)

bStarted := FALSE;
bMovementFound := FALSE;
bSearchMovement := TRUE;
iAlarmCount := 0;
TmpStepPos.iColumn := 1;
TmpStepPos.iRow := 1;

//core and ejector movements should be possible in "override" mode
//no matter if they are programmed in sequence or not
bIgnoreConditions := (((DeviceId.CompId = cCompCore) AND sv_bOverrideCoreSafety)) OR
                     (((DeviceId.CompId = cCompEjector) AND sv_bOverrideEjectorSafety));

WHILE bSearchMovement DO

   //search for the requested movement
   abInterpreter.aFindLabel.SearchStartPos := TmpStepPos;
   abInterpreter.aFindLabel(DeviceId := DeviceId, MoveId :=MoveId, MoveDir := MoveDir, IntermediateCond := IntermediateCond, bAllowNonMatchingId := FALSE);
   IF abInterpreter.aFindLabel.bFound THEN
      bMovementFound := TRUE;
      StepPos := abInterpreter.aFindLabel.StepPos;
   ELSE
      //movement not found in sequence
      bSearchMovement := FALSE;
      StepPos.iColumn := 0;
      StepPos.iRow := 0;
   END_IF;

   IF abInterpreter.aFindLabel.bFound OR NOT bNeedCheckSafety OR bIgnoreConditions THEN
      //check conditions for this movement
      abODCCheckDependenciesStart.aCheck(StepPos := StepPos, DeviceIdSelf := DeviceId, bNoAlarmsAndStepState := TRUE);

      // check existing start conditions and check conditions for the requested movement
      // attention: check is only necessary if sequence is programmed by editor
      bStartConditionOk := TRUE;
      bCheckConditionsOk := TRUE;
      bCheckConditionFound := FALSE;

      IF NOT bIgnoreConditions THEN
         IF NOT sv_bUseProgramSwitches AND bNeedCheckSafety AND abInterpreter.aFindLabel.bFound THEN
            aStartAndCheckConditions(StepPos := StepPos,
                                     bNoAlarms := TRUE,
                                     bStartConditionOk => bStartConditionOk,
                                     bCheckConditionsOk => bCheckConditionsOk,
                                     bCheckConditionFound => bCheckConditionFound);
         END_IF;
      END_IF;

      iTmpAlarmCount := 0;
      IF NOT abODCCheckDependenciesStart.aCheck.bAllowed THEN
         //safety conditions not ok => save number of not fulfilled conditions
         iTmpAlarmCount := abODCCheckDependenciesStart.aCheck.iNotOkCount;
      END_IF;

      IF NOT bStartConditionOk THEN
         //start conditions not ok => increment nummber of not fulfilled conditions
         iTmpAlarmCount := iTmpAlarmCount + aStartAndCheckConditions.iStartConditionsNotOk;
      END_IF;

      IF NOT bCheckConditionsOk THEN
         //check conditions not ok => increment nummber of not fulfilled conditions
         iTmpAlarmCount := iTmpAlarmCount + aStartAndCheckConditions.iCheckConditionsNotOk;
      END_IF;

      //everything OK -> start movement and exit loop
      IF abODCCheckDependenciesStart.aCheck.bAllowed AND bStartConditionOk AND bCheckConditionsOk THEN
         //movement with correct condition found => start this movement
         abInterpreter.aAddStartedManualMovement(DeviceId := DeviceId, MoveId := MoveId, MoveDir := MoveDir,
                                                 StepPos := StepPos, iInstance := IntermediateCond);
         IF abInterpreter.aAddStartedManualMovement.bOK THEN
            fbStart(DeviceId := DeviceId, MoveDir := MoveDir, MoveId := MoveId, IntermediateCond := IntermediateCond);
            bStarted := TRUE;

            //set step state to active
            IF (StepPos.iColumn <> 0) AND (StepPos.iRow <> 0) THEN
               fbSetStepState(StepPos := StepPos,
                              StepState := nStateActive);
            END_IF;
         END_IF;

         IF bCheckConditionFound THEN
            START_PROCESS_ALGORITHM(paCheckConditionsManual);
         END_IF;

         IF NOT abInterpreter.aFindLabel.bFound THEN
            fbDebugTrace2(nODCInterpreter, 'Manual Movement started anyway because it is not safety relevant');
         END_IF;

         bSearchMovement := FALSE;
         bMovementAllowed := TRUE;
         RETURN; // ******  exit algorithm *******
      ELSE
         //check number of not fulfilled conditions
         IF (iAlarmCount = 0) OR (iTmpAlarmCount < iAlarmCount) THEN
            //save this step
            StepPosLowestAlarms := StepPos;
            iAlarmCount := iTmpAlarmCount;
            iTmpAlarmCount := 0;
         END_IF;

         //save this position (needed as startposition of next search)
         //attention: iColumn must be increased otherwise always the same step will be found
         TmpStepPos.iColumn := StepPos.iColumn + 1;
         TmpStepPos.iRow := StepPos.iRow;
         bMovementAllowed := FALSE;
      END_IF;
   END_IF;  //end_if aFindLabel.bFound

END_WHILE;

IF NOT bMovementFound THEN
   fbDebugTrace2(nODCInterpreter, 'Manual Movement not started because movement is safety relevant but not in ODC');
ELSIF NOT bMovementAllowed THEN
   //use step which causes the lowest number of alarms
   //call dependency check again to set the according alarms
   abODCCheckDependenciesStart.aCheck(StepPos := StepPosLowestAlarms, DeviceIdSelf := DeviceId, bNoAlarmsAndStepState := FALSE);

   //set alarms related to start and check conditions
   aStartAndCheckConditions(StepPos := StepPosLowestAlarms,
                            bNoAlarms := FALSE,
                            bStartConditionOk => bStartConditionOk,
                            bCheckConditionsOk => bCheckConditionsOk,
                            bCheckConditionFound => bCheckConditionFound);

   //set step state to error
   fbSetStepState(StepPos := StepPosLowestAlarms, StepState := nStateError);

   //evCheckLocklist makes sure other alarms(caused by FBLockUnlock for this movement are also set *)
   fbDebugTrace2(nODCInterpreter, CONCAT('Manual Movement ', DINT_TO_STRING(MoveId),
                                          '/', DINT_TO_STRING(MoveDir),
                                          ' not started because safety conditions do not allow it -> sending evCheckLocklist to view all other alarms'));
   evCheckLocklistEventData.DeviceId := DeviceId;
   evCheckLocklistEventData.MoveId   := MoveId;
   evCheckLocklistEventData.MoveDir  := MoveDir;
   SET_EVENT(evCheckLocklist, evCheckLocklistEventData);

   IF NOT bStartConditionOk THEN
      fbDebugTrace2(nODCInterpreter, 'Manual Movement not started because start condition not ok');
   END_IF;

   IF NOT bCheckConditionsOk THEN
      fbDebugTrace2(nODCInterpreter, 'Manual Movement not started because check condition not ok');
   END_IF;
END_IF;

@END_Body

@@@BEG_Comment@@@
@TL(11)
Start a single movement (in response to evStartRequest)

Basically the same movement can occur more than one time in the machine sequence.
If the requested movement is found in the sequence and all conditions are ok, this movement is started.
If one or more conditions (safety conditions, start conditions, check conditions) are not ok, the
algorithm continues searching because possibly the movement is found again and the conditions for this step are ok.

If the movement is not allowed, the movement position with the lowest number of not fulfilled conditions is marked (step state is set)
and tha according alarms are set

@@@END_Comment@@@

@BEG_Body
@TL(56)
(**************************************** WARNING ********************************************
 *** The KEBA Kemro K2 System including software is not intended for safety control tasks! ***
 ***                       For further information see Comment tab!                        ***
 *********************************************************************************************)

bNotFound := FALSE;

(* find start label *)
abInterpreter.aFindLabel.SearchStartPos.iColumn := 1;
abInterpreter.aFindLabel.SearchStartPos.iRow := 1;
abInterpreter.aFindLabel(DeviceId := DeviceId,
                         MoveId := cMoveBeginSequence,
                         MoveDir := MoveDir,
                         IntermediateCond := 0,
                         bAllowNonMatchingId := FALSE);
IF NOT abInterpreter.aFindLabel.bFound THEN
   fbDebugTrace2(nODCInterpreter, 'combined movement -> start label not found -> will try to start single movement');
   bNotFound := TRUE;
   RETURN;
END_IF;

StartPos := abInterpreter.aFindLabel.StepPos;

(* find end of label *)
abInterpreter.aFindLabel(DeviceId := DeviceId,
                         MoveId := cMoveEndSequence,
                         MoveDir := MoveDir,
                         IntermediateCond := 0,
                         bAllowNonMatchingId := FALSE);
IF NOT abInterpreter.aFindLabel.bFound THEN
   fbDebugTrace2(nODCInterpreter, 'combined movement -> end label not found -> will try to start single movement');
   bNotFound := TRUE;
   RETURN;
END_IF;

// save active sequence (for highlighting in machine sequencer)
sv_ActiveSequence.DeviceId := DeviceId;
sv_ActiveSequence.MoveDir := MoveDir;
sv_ActiveSequence.iCount :=  sv_ActiveSequence.iCount + 1;
sv_ActiveSequence.bActive := TRUE;

(* remember for later so we can stop combined movements *)
mStartedCombinedMovement.DeviceId := DeviceId;
mStartedCombinedMovement.MoveId   := MoveId;
mStartedCombinedMovement.MoveDir  := MoveDir;

abInterpreter.aInitInterpreter(iColumn := StartPos.iColumn,
                               iRow := StartPos.iRow,
                               iEndRow := abInterpreter.aFindLabel.StepPos.iRow,
                               bSkipAlreadyPosReached := TRUE,
                               bExcludeActiveColumns := FALSE);

(* paRunManualCombinedMovement stops itself when interpreter is not active anymore *)
START_PROCESS_ALGORITHM(paRunManualCombinedMovement);

@END_Body

@@@BEG_Comment@@@
@TL(1)
Start a combined movement (in response to evStartRequest)
@@@END_Comment@@@

@BEG_Body
@TL(180)
(**************************************** WARNING ********************************************
 *** The KEBA Kemro K2 System including software is not intended for safety control tasks! ***
 ***                       For further information see Comment tab!                        ***
 *********************************************************************************************)

IF mbRecalcActive THEN
   //Ignore start requests if a cycle recalc is active.
   //This flag is set by aDoPendingRecalc() before the low priority paInitSequence actually starts executing code
   //This is necessary to avoid problems where a recalc and a movement start happen at the same cycle
   fbDebugTrace2(nDeviceState, 'evStartRequest ignored because sequence is being recalculated');
   RETURN;
END_IF;

IF sv_iInitOK <> 20 THEN
   //ignore start requests if array is not initialized completely
   //this can happen during startup and during creation of a new sequence
   //or if creation of a sequence failed
   fbDebugTrace2(nDeviceState, 'evStartRequest ignored because sequence not initialized');
   RETURN;
END_IF;

IF sv_OperationMode >= nHalfAutomatic THEN
   IF sv_bSequenceInterruption THEN
      //sequence is actually interrupted -> find out if it is allowed to start this movement
      fbGetMoveNumber(DeviceId := evStartRequestData.DeviceId,
                     MoveDir := evStartRequestData.MoveDir,
                     MoveId := evStartRequestData.MoveId);

      IF fbGetMoveNumber.bFound THEN
         IF sv_MovementsAvailable[fbGetMoveNumber.iMoveNumber].pMovementData^.bAllowedDuringInterrupt THEN
            //try to start this movement
            aStartSingleMovement(DeviceId := evStartRequestData.DeviceId,
                                 MoveDir := evStartRequestData.MoveDir,
                                 MoveId := evStartRequestData.MoveId,
                                 IntermediateCond := evStartRequestData.IntermediateCond,
                                 bNeedCheckSafety := FALSE);
         END_IF;
      END_IF;
   ELSE
      //ignore start requests if operation mode is half or full automatic
      fbDebugTrace2(nDeviceState, 'evStartRequest ignored because in half or full auto mode');
   END_IF;

   RETURN; // return here
END_IF;

IF sv_iActiveEditors > 0 THEN
   //teach mode active -> ignore start requests
   SET_ALARM(Name := erTeachModeActive);
   RETURN;
END_IF;

StartRequestData := evStartRequestData;

// work with StartRequest
fbGetMoveNumber(DeviceId := StartRequestData.DeviceId,
                MoveDir := StartRequestData.MoveDir,
                MoveId := StartRequestData.MoveId);

IF fbGetMoveNumber.bFound THEN
   iSafety := sv_MovementsAvailable[fbGetMoveNumber.iMoveNumber].pMovementData^.iSafetyIdentifier;
   (* FIXME: always set the intermediate condition to 0 when movement does not have intermediate conditions
      needed for searching the movement
   *)
   IF NOT sv_MovementsAvailable[fbGetMoveNumber.iMoveNumber].pMovementData^.bInstanceable THEN
      StartRequestData.IntermediateCond := 0;
   END_IF;
ELSE
   fbDebugTrace2(nODCInterpreter, 'could not find movement -> assuming movement is safety relevant');
   iSafety := 1;
END_IF;

IF iSafety = 1 THEN
   bCheckSafety := TRUE;
   fbDebugTrace2(nODCInterpreter, 'movement is safety relevant (sequence safety and mold safety (safety editor)');
ELSIF iSafety = 3 THEN
   bCheckSafety := TRUE;
   fbDebugTrace2(nODCInterpreter, 'movement is safety relevant (sequence safety only - no mold safety (safety editor)');
ELSIF iSafety = 2 THEN
   // only check pos reached of other movements, movement itself is not safety relevant
   bCheckSafety := TRUE;
   fbDebugTrace2(nODCInterpreter, 'movement is partially safety relevant');
ELSIF iSafety = 0 THEN
   bCheckSafety := FALSE;
   fbDebugTrace2(nODCInterpreter, 'movement is NOT safety relevant');
ELSE
   bCheckSafety := TRUE;
   fbDebugTrace(CONCAT('strange safety relevance value ', DINT_TO_STRING(iSafety)));
END_IF;

abInterpreter.aStatus();
IF abInterpreter.aStatus.bActive THEN
   fbDebugTrace2(nODCInterpreter, 'manual movement not started because there is already a combined movement active');

   SET_ALARM(Name := erMovementDuringActiveSequence,
             SubID1 := StartRequestData.DeviceId.CompId,
             SubID2 := StartRequestData.MoveId,
             SubID3 := mStartedCombinedMovement.DeviceId.CompId,
             SubID4 := mStartedCombinedMovement.MoveId,
             Param1 := DINT_TO_STRING(StartRequestData.DeviceId.IndexId));
   RETURN;
END_IF;

(* Rules:
 * When a combined movement is active no other movement may be started
 * When any movement is active no combined movement may be started
 * Autopurge counts as 1 or more movementy so the above rule covers this already
   -> single movements are allowed during autopurge
 * When operation mode is setup, combined movement are never started(only single movemets *)

IF sv_bCombinedMovementsInManual AND (StartRequestData.MoveId = cMoveBeginSequence) THEN
   IF sv_OperationMode = nSetup THEN
      fbDebugTrace2(nODCInterpreter, 'starting a combined movement in setup mode is not allowed');
      RETURN;
   END_IF;
   bCombined := TRUE;
ELSIF sv_bCombinedMovementsInManual AND (sv_OperationMode = nManual) AND
   (* combined movements are not allowed in setup mode *)
   (StartRequestData.DeviceId.CompId = cCompMold AND
   ((StartRequestData.MoveDir = cMoveFwd OR
    StartRequestData.MoveDir = cMoveBwd))
   OR
   (StartRequestData.DeviceId.CompId = cCompInjection AND
   (StartRequestData.MoveId = cMoveInject OR
    StartRequestData.MoveId = cMoveCombinedPlast))) THEN
   //this check is for MoveId as plasticize, decompress and intrusion have MoveDir = cMoveBwd
   bCombined := TRUE;
ELSE
   bCombined := FALSE;

   //check if  requested device is activated
   FOR i := 1 TO sv_ODCDeviceMovements.iCount DO
      IF sv_ODCDeviceMovements.Devices[i].DeviceId = StartRequestData.DeviceId THEN
         IF NOT sv_ODCDeviceMovements.Devices[i].pbDeviceActivated^ THEN
            fbDebugTrace2(nODCInterpreter, 'start request ignored because device is not activated');
            RETURN;
         END_IF;
         EXIT;
      END_IF;
   END_FOR;
END_IF;

IF sv_StartedMovements.iStartedMovements <> 0 AND bCombined THEN
   fbDebugTrace2(nODCInterpreter, 'combined manual movement not started because there is already a movement active');

   SET_ALARM(Name := erSequenceDuringActiveMovement,
             SubID1 := StartRequestData.DeviceId.CompId,
             SubID2 := StartRequestData.DeviceId.IndexId,
             SubID3 := StartRequestData.MoveId);
   RETURN;
END_IF;

(* back up sequence when a movement is started
   and the sequence has changed *)
START_PROCESS_ALGORITHM(paBackupSequence);

IF bCombined THEN
   fbDebugTrace2(nODCInterpreter, 'evStartRequest -> starting a combined movement');
   aClearStepState(FALSE);
   aStartCombinedMovement(DeviceId := StartRequestData.DeviceId,
                          MoveDir := StartRequestData.MoveDir,
                          MoveId := StartRequestData.MoveId);
END_IF;

IF NOT bCombined OR aStartCombinedMovement.bNotFound THEN
   (* if combined movement markers were not found start single movement *)
   IF (StartRequestData.MoveId = cMoveBeginSequence) THEN
      //do not try to start a single movement if a start request for
      //cMoveBeginSequence was received and this sequence was not found
      fbDebugTrace2(nODCInterpreter, 'requested combined movement not found');
   ELSE
      fbDebugTrace2(nODCInterpreter, 'evStartRequest -> starting a single movement');
      aStartSingleMovement(DeviceId := StartRequestData.DeviceId,
                           MoveDir := StartRequestData.MoveDir,
                           MoveId := StartRequestData.MoveId,
                           IntermediateCond := StartRequestData.IntermediateCond,
                           bNeedCheckSafety := bCheckSafety);
   END_IF;
END_IF;

@END_Body

@@@BEG_Comment@@@
@TL(6)
Handle evStartRequest(manual buttons)
start requests will be ignored in the following situations:
- sequence array not initialized completely
  (startup or creation of new sequence in progress, creation of sequence failed)
- machine running in half or fullauto cycle
- teachmode in machine sequencer is active
@@@END_Comment@@@

@BEG_Body
@TL(49)
(**************************************** WARNING ********************************************
 *** The KEBA Kemro K2 System including software is not intended for safety control tasks! ***
 ***                       For further information see Comment tab!                        ***
 *********************************************************************************************)

IF NOT sv_bInitDone THEN
   //ignore stop requests before sv_bInitDone
   fbDebugTrace2(nDeviceState, 'evStopRequest ignored because sv_bInitDone is not TRUE');
   RETURN;
END_IF;

IF (sv_OperationMode >= nHalfAutomatic) AND NOT sv_bSequenceInterruption THEN
   //ignore stop requests if operation mode is half or full automatic
   //stop requests for movements which were started during sequence interruption
   //must be handled
   fbDebugTrace2(nDeviceState, 'evStopRequest ignored because in half or full auto mode');
   RETURN;
END_IF;

abInterpreter.aStatus();
IF abInterpreter.aStatus.bActive THEN
   IF mStartedCombinedMovement.DeviceId = evStopRequestData.DeviceId AND
      mStartedCombinedMovement.MoveId = evStopRequestData.MoveId AND
      mStartedCombinedMovement.MoveDir = evStopRequestData.MoveDir THEN
      // we get a stop request for the combined movement
      // so stop it
      fbDebugTrace2(nDeviceState, 'evStopRequest while interpreter is active -> aStopInterpreterNormal()');
      abInterpreter.aStopInterpreterNormal();
      sv_ActiveSequence.bActive := FALSE;
   ELSE
      // we get a stop request for a single movement
      // but a combined movement is active
      // but no single movements are allowed during a combined movement
      // -> ignore the event
      fbDebugTrace2(nDeviceState, 'evStopRequest ignored because combined movement is active and device/movement does not match');
   END_IF;
ELSE
   fbDebugTrace2(nDeviceState, 'evStopRequest while interpreter is inactiveactive -> fbStop()');
   // it is also possible that the interpreter already finished the combined movement
   // we still send a evStop, but that does not cause ony problems
   fbStop(DeviceId := evStopRequestData.DeviceId);
   sv_ActiveSequence.bActive := FALSE;
END_IF;

// no movenumber available, clear all
g_SafetyData.MovementToActivate := 0;

@END_Body

@@@BEG_Comment@@@
@TL(2)
Handle evStopRequest(manual buttons)
Stop single and combined movements
@@@END_Comment@@@

@BEG_Body
@TL(43)
(**************************************** WARNING ********************************************
 *** The KEBA Kemro K2 System including software is not intended for safety control tasks! ***
 ***                       For further information see Comment tab!                        ***
 *********************************************************************************************)

FOR i := 1 TO sv_iUsedColumns DO
   IF (mActiveStepBwdMovements[i].DeviceId = DeviceId) AND
      (mActiveStepBwdMovements[i].MoveId = MoveId) AND
      (mActiveStepBwdMovements[i].MoveDir = MoveDir) THEN

      //check posReached flag
      fbCheckPosReached(DeviceId := DeviceId,
                        MoveDir := MoveDir,
                        MoveId := MoveId);

      IF CHECK_REF(fbCheckPosReached.pbPosReached^) AND NOT fbCheckPosReached.pbPosReached^ THEN
         ;//endposition not reached -> do not decrease line number
      ELSE
         //endposition reached or no posReached flag available -> decrease row
         iTmpColumn := i;
         REPEAT
            IF sv_TraceLevel.bODCInterpreter THEN
               dummy := Print('call abInterpreter.aDecreaseRow with iColumn = %d', iTmpColumn);
            END_IF;
            abInterpreter.aDecreaseRow(bStartInActualLine := FALSE,
                                       iColumn := iTmpColumn,
                                       iEndRow := 1);
            iTmpColumn := abInterpreter.aDecreaseRow.iNewActivatedColumn;

         UNTIL (abInterpreter.aDecreaseRow.iNewActivatedColumn = 0)
         END_REPEAT;
      END_IF;

      //init this element
      mActiveStepBwdMovements[i].DeviceId.CompId := cCompNone;
      mActiveStepBwdMovements[i].DeviceId.IndexId := 1;
      mActiveStepBwdMovements[i].MoveId := cMinMoveIdent;
      mActiveStepBwdMovements[i].MoveDir := cMoveNone;

      EXIT;
   END_IF;
END_FOR;

@END_Body

@@@BEG_Comment@@@
@TL(0)

@@@END_Comment@@@

@BEG_Body
@TL(91)
(**************************************** WARNING ********************************************
 *** The KEBA Kemro K2 System including software is not intended for safety control tasks! ***
 ***                       For further information see Comment tab!                        ***
 *********************************************************************************************)

IF evStartedStoppedData.State = nStopped OR  evStartedStoppedData.State = nStartNotAllowed THEN
   bFound := FALSE;
   // movement was stopped or never started
   // remove movement from list with started movements

   Status := MovementsSema.Wait(WaitTime := cTimeOutSempahore);
   IF Status <> KRTOS_Status_OK THEN
      dummy2 := ASSERT(FALSE, erAssert);
      RETURN;
   END_IF;

   FOR i := 1 TO sv_StartedManualMovements.iStartedMovements DO

      bCorrectInstance := (evStartedStoppedData.iInstance = 0) OR (evStartedStoppedData.iInstance = sv_StartedManualMovements.MoveData[i].iInstance);
      IF sv_StartedManualMovements.MoveData[i].DeviceId = evStartedStoppedData.DeviceId AND
         sv_StartedManualMovements.MoveData[i].MoveDir = evStartedStoppedData.MoveDir AND
         sv_StartedManualMovements.MoveData[i].MoveId = evStartedStoppedData.MoveId AND bCorrectInstance THEN

         stepPos := sv_StartedManualMovements.MoveData[i].StepPos;
         IF (g_SafetyData.bAvailable) THEN
            IF (NOT((stepPos.iColumn = 0) OR (stepPos.iRow = 0)))THEN
               idx := sv_MovementsAvailable[sv_ODCSequenceInt[stepPos.iColumn][stepPos.iRow].iMoveNumber].iODCSafetyMovementsEntry;
               IF (idx > 0) THEN
                  g_SafetyData.MovementToActivate := g_SafetyData.MovementToActivate AND (NOT SHL(1, idx-1));
               END_IF;
            END_IF;
         END_IF;

         IF (NOT((stepPos.iColumn = 0) OR (stepPos.iRow = 0)))THEN
            //only correct step sate if actual state is not error
            IF sv_ODCSequenceInt[stepPos.iColumn, stepPos.iRow].StepState <> nStateError THEN
               fbSetStepState(StepPos := sv_StartedManualMovements.MoveData[i].StepPos,
                           StepState := nStateReady);
            END_IF;

         END_IF;

         IF sv_TraceLevel.bODCInterpreter THEN
            dummy := Print('removing started manual movement %d.%d %d/%d', evStartedStoppedData.DeviceId.CompId, evStartedStoppedData.DeviceId.IndexId, evStartedStoppedData.MoveId, evStartedStoppedData.MoveDir);
         END_IF;

         //copy last entry in the list to this empty field
         sv_StartedManualMovements.MoveData[i] := sv_StartedManualMovements.MoveData[sv_StartedManualMovements.iStartedMovements];

         //zero last entry
         tmpMovement.DeviceId.CompId := cCompNone;
         tmpMovement.DeviceId.IndexId := 1;
         tmpMovement.MoveDir := cMoveNone;
         tmpMovement.MoveId := cMinMoveIdent;
         tmpMovement.StepPos.iColumn := 0;
         tmpMovement.StepPos.iRow := 0;
         tmpMovement.iInstance := 0;
         sv_StartedManualMovements.MoveData[sv_StartedManualMovements.iStartedMovements] := tmpMovement;

         sv_StartedManualMovements.iStartedMovements := sv_StartedManualMovements.iStartedMovements - 1;
         //fbDebugTrace2(nODCInterpreter, 'end removing started manual movement');
         bFound := TRUE;
         EXIT;
      END_IF;
   END_FOR;

   Status := MovementsSema.Put();
   IF Status <> KRTOS_Status_OK THEN
      dummy2 := ASSERT(FALSE, erAssert);
   END_IF;

   IF sv_bSequenceInterruption THEN
      //started / stopped event during sequence is interrupted
      //-> check if line number should be decreased
      aDecreaseLineNumber(DeviceId := evStartedStoppedData.DeviceId,
                          MoveId := evStartedStoppedData.MoveId,
                          MoveDir := evStartedStoppedData.MoveDir);
   END_IF;

   IF NOT bFound THEN
      IF sv_TraceLevel.bODCInterpreter THEN
         dummy := Print('tried to remove stopped movement, but not in list anymore???');
      END_IF;
   END_IF;
END_IF;

@END_Body

@@@BEG_Comment@@@
@TL(2)
Manage list and count of currently started movments
in sv_StartedMovements when receiving evStartedStopped events
@@@END_Comment@@@

@BEG_Body
@TL(22)
(**************************************** WARNING ********************************************
 *** The KEBA Kemro K2 System including software is not intended for safety control tasks! ***
 ***                       For further information see Comment tab!                        ***
 *********************************************************************************************)

IF sv_StartedManualMovements.iStartedMovements = 0 THEN
   STOP_PROCESS_ALGORITHM(paCyclicConditionCheck);
   STOP_PROCESS_ALGORITHM(paCheckConditionsManual);

   abInterpreter.aStatus();
   IF sv_OperationMode <= nManual AND NOT abInterpreter.aStatus.bActive THEN
      (* the last single manual movement was stopped -> recalculate if needed *)
      aDoPendingRecalc();
      IF aDoPendingRecalc.bStartedRecalc THEN
         fbDebugTrace2(nDeviceState, 'recalc because iStartedMovements = 0');
      END_IF;
   END_IF;
ELSE
   START_PROCESS_ALGORITHM(paCyclicConditionCheck);

END_IF;

@END_Body

@@@BEG_Comment@@@
@TL(2)
Start / stop paCyclicConditionCheck depending on
if there are started movements.
@@@END_Comment@@@

@BEG_Body
@TL(43)
(**************************************** WARNING ********************************************
 *** The KEBA Kemro K2 System including software is not intended for safety control tasks! ***
 ***                       For further information see Comment tab!                        ***
 *********************************************************************************************)

abInterpreter.aStatus();

Status := MovementsSema.Wait(WaitTime := cTimeOutSempahore);
IF Status <> KRTOS_Status_OK THEN
   dummy2 := ASSERT(FALSE, erAssert);
   RETURN;
END_IF;

FOR i := 1 TO sv_StartedManualMovements.iStartedMovements DO
   // check safety for manual movements
   // abODCCheckSafetyConditions must be a separete instance
   // because this PROCESS_ALGORITHM runs in a fast task that can
   // interrupt other tasks
   TmpStepPos := sv_StartedManualMovements.MoveData[i].StepPos;
   IF(abInterpreter.aStatus.bActive AND (TmpStepPos.iColumn = 0 OR TmpStepPos.iRow = 0)) THEN
      fbDebugTrace('interpreter is active but a movement with step pos 0 is running'); //this might be legitime, but is most times not normal
      abInterpreter.aStopInterpreterFatal();
   END_IF;

   abODCCheckDependenciesCyclic.aCheck(StepPos := TmpStepPos, DeviceIdSelf := sv_StartedManualMovements.MoveData[i].DeviceId);
   IF NOT abODCCheckDependenciesCyclic.aCheck.bAllowed THEN
      fbDebugTrace2(nODCInterpreter, CONCAT('cyclic condition check reported movement at ',
                                            DINT_TO_STRING(sv_StartedManualMovements.MoveData[i].StepPos.iColumn),
                                            '/',
                                            DINT_TO_STRING(sv_StartedManualMovements.MoveData[i].StepPos.iRow),
                                            ' as not allowed'));
      abInterpreter.aStopInterpreterError();
   END_IF;

END_FOR;

//FIXME: is it a good idea to hold the lock so long???
Status := MovementsSema.Put();
IF Status <> KRTOS_Status_OK THEN
   dummy2 := ASSERT(FALSE, erAssert);
END_IF;

@END_Body

@@@BEG_Comment@@@
@TL(2)
Cyclically check movement conditions of all started movements
(auto mode, combined manual movements, single manual movements)
@@@END_Comment@@@

@BEG_SfcBody
80 46 55

@BEG_SfcData 2
@StepSeq @RT(4)sseq @F 3
@Step @RT(16)S_CheckStartCond @F @T @T @F @RT(0) @F
@AcbCont @RT(7)unnamed @F 1
@Acb @RT(15)AAutoCycleReady @F @T @RT(1)P @RT(0) @F @F @T @TL(7)
bReady := TRUE;
IF (sv_OperationMode <> nFullAutomatic) THEN
   sv_bAutoCycleRunning := FALSE;
END_IF;
g_SafetyData.MovementToActivate := 0;
abInterpreter.aResetStepMode();

@F

@Trans @RT(13)T_StartCondOK @F @T @F @F @T @F @TL(2)
NOT bStopCycle AND NOT bStopAfterCycle

@RT(6)Trans1 @F
@Loop @RT(4)loop @F 2
@StepSeq @RT(3)seq @F 9
@Loop @RT(4)loop @F 2
@StepSeq @RT(3)seq @F 13
@Step @RT(17)S_CheckStartCycle @F @F @T @F @RT(0) @F
@AcbCont @RT(7)unnamed @F 4
@Acb @RT(9)AAutoInit @F @T @RT(1)P @RT(0) @F @F @T @TL(7)
bReady := FALSE;
IF (sv_OperationMode <> nFullAutomatic) THEN
   sv_bAutoCycleRunning := FALSE;
END_IF;
bCanStart := FALSE;
abWaitCycleStart.aCycleStartRequest();

@F
@Acb @RT(15)AWaitCycleStart @F @T @RT(1)N @RT(0) @F @F @T @TL(6)
abWaitCycleStart.aWaitCycleStart();
IF abWaitCycleStart.aWaitCycleStart.bCanStart THEN
   (* save flag because it is only TRUE for 1 cycle *)
   bCanStart := TRUE;
END_IF;

@F
@Acb @RT(7)aRecalc @F @T @RT(1)N @RT(0) @F @F @T @TL(7)
// allow to recalculate the cycle while waiting for the start signal
// but delay real start of the sequence until recalculation is finished
aDoPendingRecalc();
IF aDoPendingRecalc.bStartedRecalc THEN
   fbDebugTrace2(nDeviceState, 'recalc because autocycle start wait');
END_IF;

@F
@Acb @RT(11)ADelayCycle @F @F @RT(1)N @RT(0) @F @F @F @F

@Trans @RT(12)T_StartCycle @F @T @F @F @T @F @TL(2)
bCanStart AND bDelayExceeded AND NOT mbRecalcActive

@RT(6)Trans2 @F
@Step @RT(6)Step42 @F @F @F @F @RT(0) @F
@AcbCont @RT(7)unnamed @F 0

@AltBranch @RT(3)alt @F 2
@TransSeq @RT(4)tseq @F 3
@Trans @RT(20)TSequenceInterrupted @F @T @F @F @T @F @TL(2)
sv_bSequenceInterruption

@RT(7)Trans48 @F
@Step @RT(6)Step43 @F @F @F @F @RT(0) @F
@AcbCont @RT(7)unnamed @F 0

@AltBranch @RT(3)alt @F 2
@TransSeq @RT(4)tseq @F 1
@Trans @RT(17)TContinueSequence @F @T @F @F @T @T @TL(2)
NOT sv_bSequenceInterruption

@RT(7)Trans50 @F

@TransSeq @RT(4)tseq @F 4
@Trans @RT(7)Trans51 @F @T @F @F @T @T @TL(2)
di_StepFwd

@RT(7)Trans51 @F
@Step @RT(6)Step44 @F @F @F @F @RT(0) @F
@AcbCont @RT(7)unnamed @F 1
@Acb @RT(25)AMovementsBeforeCycleLoop @F @T @RT(1)P @RT(0) @F @F @T @TL(6)
IF (g_iAutoCycleLoopStartLine > 2) THEN
   bMovesBeforeAutoLoop := TRUE;
ELSE
   bMovesBeforeAutoLoop := FALSE;
END_IF;

@F

@AltBranch @RT(3)alt @F 2
@TransSeq @RT(4)tseq @F 1
@Trans @RT(21)TMovementsBeforeCycle @F @T @F @F @T @F @TL(2)
bMovesBeforeAutoLoop

@RT(7)Trans52 @F

@TransSeq @RT(4)tseq @F 2
@Trans @RT(22)TNoMoveBeforeAutocycle @F @T @F @F @T @F @TL(3)
NOT bMovesBeforeAutoLoop

@RT(7)Trans53 @F
@Goto @RT(6)S_ODC1 @F @F

@Goto @RT(17)S_BeforeCycleLoop @F @F

@TransSeq @RT(4)tseq @F 1
@Trans @RT(7)Trans49 @F @T @T @F @T @F @TL(2)
NOT sv_bSequenceInterruption

@RT(7)Trans49 @F

@Step @RT(6)Step20 @F @F @F @F @RT(0) @F
@AcbCont @RT(7)unnamed @F 0

@AltBranch @RT(3)alt @F 2
@TransSeq @RT(4)tseq @F 5
@Trans @RT(11)TFirstCycle @F @T @F @F @T @F @TL(2)
sv_bFirstCycle

@RT(7)Trans19 @F
@Step @RT(16)S_EjectorAutoBwd @F @F @F @F @RT(0) @F
@AcbCont @RT(7)unnamed @F 2
@Acb @RT(15)AInitEjectorBwd @F @F @RT(1)P @RT(0) @F @F @F @F
@Acb @RT(15)AEjectorAutoBwd @F @F @RT(1)P @RT(0) @F @F @F @F

@AltBranch @RT(3)alt @F 2
@TransSeq @RT(4)tseq @F 3
@Trans @RT(15)TEjectorStarted @F @T @F @F @T @F @TL(2)
bEjectorBwdStarted AND pbEjectorReady^

@RT(7)Trans12 @F
@Step @RT(17)S_CheckEjectorBwd @F @F @F @F @RT(0) @F
@AcbCont @RT(7)unnamed @F 1
@Acb @RT(16)ACheckEjectorBwd @F @F @RT(1)P @RT(0) @F @F @F @F

@Trans @RT(11)TEjectorBwd @F @T @F @F @T @F @TL(2)
pbEjectorBwd^

@RT(7)Trans10 @F

@TransSeq @RT(4)tseq @F 1
@Trans @RT(18)TEjectorNotStarted @F @T @T @F @T @F @TL(2)
NOT bEjectorBwdStarted

@RT(7)Trans13 @F

@Step @RT(17)S_BeforeCycleLoop @F @F @T @F @RT(0) @F
@AcbCont @RT(7)unnamed @F 2
@Acb @RT(17)AStepsBeforeCycle @F @T @RT(1)P @RT(0) @F @F @T @TL(10)
aClearStepState(FALSE);
abInterpreter.aInitInterpreter(iColumn := 1,
                               iRow := 1,
                               iEndRow := g_iAutoCycleLoopStartLine,
                               bSkipAlreadyPosReached := FALSE,
                               bExcludeActiveColumns := FALSE);

abInterpreter.aIncreaseRow(iColumn := 1,
                           iEndRow := g_iAutoCycleLoopStartLine);

@F
@Acb @RT(20)ARunStepsBeforeCycle @F @T @RT(1)N @RT(0) @F @F @T @TL(3)
abInterpreter.aInterpret();
abInterpreter.aStatus();

@F

@Trans @RT(17)TBeforeCycleReady @F @T @F @F @T @T @TL(2)
abInterpreter.aStatus.bFinished

@RT(7)Trans17 @F

@TransSeq @RT(4)tseq @F 2
@Trans @RT(14)TNotFirstCycle @F @T @F @F @T @F @TL(2)
NOT sv_bFirstCycle

@RT(7)Trans42 @F
@Goto @RT(6)S_ODC1 @F @F

@Step @RT(6)S_ODC1 @F @F @T @F @RT(0) @F
@AcbCont @RT(7)unnamed @F 2
@Acb @RT(11)AStartCycle @F @F @RT(1)P @RT(0) @F @F @F @F
@Acb @RT(16)AInitInterpreter @F @F @RT(1)P @RT(0) @F @F @F @F

@Trans @RT(7)Trans32 @F @T @F @F @T @F @TL(2)
TRUE

@RT(7)Trans32 @F
@Step @RT(5)S_Run @F @F @F @F @RT(0) @F
@AcbCont @RT(7)unnamed @F 1
@Acb @RT(15)ARunInterpreter @F @T @RT(1)N @RT(0) @F @F @T @TL(3)
abInterpreter.aInterpret();
abInterpreter.aStatus();

@F

@AltBranch @RT(3)alt @F 2
@TransSeq @RT(4)tseq @F 1
@Trans @RT(13)T_ODCFinished @F @T @F @F @T @F @TL(2)
abInterpreter.aStatus.bFinished

@RT(7)Trans17 @F

@TransSeq @RT(4)tseq @F 4
@Trans @RT(10)T_ODCError @F @T @F @F @T @F @TL(2)
abInterpreter.aStatus.bError

@RT(6)Trans3 @F
@Step @RT(10)SErrorWait @F @F @F @F @RT(0) @F
@AcbCont @RT(7)unnamed @F 1
@Acb @RT(11)AAutoManual @F @T @RT(1)N @RT(0) @F @F @T @TL(2)
fbAutoManual();

@F

@Trans @RT(5)TStop @F @T @F @F @T @T @TL(2)
bStopCycle

@RT(6)Trans4 @F
@Goto @RT(16)S_CheckStartCond @F @F

@Step @RT(13)S_FinishCycle @F @F @F @F @RT(0) @F
@AcbCont @RT(7)unnamed @F 2
@Acb @RT(20)AIncreaseShotCounter @F @T @RT(1)P @RT(0) @F @F @T @TL(8)
g_SafetyData.MovementToActivate := 0;

fbStart.DeviceId.CompId := cCompOperationMode;
fbStart.DeviceId.IndexId := 1;
fbStart.MoveDir := cMoveNone;
fbStart.MoveId := cMoveIncreaseShotCounter;
fbStart();

@F
@Acb @RT(11)AResetFlags @F @T @RT(1)P @RT(0) @F @F @T @TL(3)
sv_bFirstCycle := FALSE;
mbCycleTimeMachineRunning := FALSE;

@F

@Trans @RT(7)Trans52 @F @T @F @F @T @T @TL(2)
TRUE

@RT(7)Trans75 @T @TL(1)
must be IEC transition because of shot counter / production counter

@Step @RT(16)S_CheckStopCycle @F @F @F @F @RT(0) @F
@AcbCont @RT(7)unnamed @F 1
@Acb @RT(19)ACheckRecalcPending @F @T @RT(1)P @RT(0) @F @F @T @TL(2)
bDoRecalc := (mPendingRecalc <> nODCRecalcNone)

@F

@Trans @RT(10)T_NewCycle @F @T @T @T @T @F @TL(3)
NOT bStopAfterCycle AND
NOT bDoRecalc

@RT(7)Trans13 @F

@Trans @RT(13)TStopOrRecalc @F @T @F @F @T @F @TL(2)
bStopAfterCycle OR bDoRecalc

@RT(7)Trans28 @F
@Step @RT(6)Step27 @F @F @F @F @RT(0) @F
@AcbCont @RT(7)unnamed @F 1
@Acb @RT(18)ACheckColumnActive @F @T @RT(1)P @RT(0) @F @F @T @TL(2)
aIsAnyColumnActive(bActive => bColumnActive);

@F

@AltBranch @RT(3)alt @F 2
@TransSeq @RT(4)tseq @F 5
@Trans @RT(7)Trans21 @F @T @F @F @T @F @TL(3)
//"parallel open" movements must also be finished
bColumnActive

@RT(7)Trans21 @F
@Step @RT(20)S_FinishParallelOpen @F @F @F @F @RT(0) @F
@AcbCont @RT(7)unnamed @F 2
@Acb @RT(19)AFinishParallelOpen @F @T @RT(1)N @RT(0) @F @F @T @TL(4)
//call interpreter until all columns
//are finished
abInterpreter.aInterpret();

@F
@Acb @RT(13)ACheckColumns @F @T @RT(1)N @RT(0) @F @F @T @TL(2)
aIsAnyColumnActive(bActive => bColumnActive);

@F

@Trans @RT(7)Trans23 @F @T @F @F @T @T @TL(2)
NOT bColumnActive

@RT(7)Trans23 @F
@Step @RT(6)Step24 @F @F @F @F @RT(0) @F
@AcbCont @RT(7)unnamed @F 0

@AltBranch @RT(3)alt @F 2
@TransSeq @RT(4)tseq @F 1
@Trans @RT(7)Trans24 @F @T @F @F @T @F @TL(2)
bStopAfterCycle

@RT(7)Trans24 @F

@TransSeq @RT(4)tseq @F 2
@Trans @RT(7)Trans27 @F @T @F @F @T @F @TL(2)
bDoRecalc

@RT(7)Trans27 @F
@Goto @RT(17)S_CheckStartCycle @F @F

@TransSeq @RT(4)tseq @F 1
@Trans @RT(7)Trans22 @F @T @T @F @T @F @TL(2)
NOT bColumnActive

@RT(7)Trans22 @F

@Step @RT(16)S_AfterCycleLoop @F @F @F @F @RT(0) @F
@AcbCont @RT(7)unnamed @F 2
@Acb @RT(16)AStepsAfterCycle @F @T @RT(1)P @RT(0) @F @F @T @TL(9)
abInterpreter.aInitInterpreter(iColumn := 1,
                               iRow := g_iAutoCycleLoopEndLine,
                               iEndRow := sv_iUsedRows,
                               bSkipAlreadyPosReached := FALSE,
                               bExcludeActiveColumns := FALSE);

abInterpreter.aIncreaseRow(iColumn := 1,
                           iEndRow := sv_iUsedRows);

@F
@Acb @RT(19)ARunStepsAfterCycle @F @T @RT(1)N @RT(0) @F @F @T @TL(3)
abInterpreter.aInterpret();
abInterpreter.aStatus();

@F

@Trans @RT(7)Trans14 @F @T @F @F @T @F @TL(2)
abInterpreter.aStatus.bFinished

@RT(7)Trans14 @F
@Step @RT(11)S_WaitReady @F @F @F @F @RT(0) @F
@AcbCont @RT(7)unnamed @F 0

@Trans @RT(18)TAllMovementsReady @F @T @F @F @T @F @TL(4)
//wait untill all movements are ready
//for example airvalve movement can be still active
sv_StartedManualMovements.iStartedMovements = 0

@RT(6)Trans8 @F
@Step @RT(5)S_End @F @F @F @F @RT(0) @F
@AcbCont @RT(7)unnamed @F 1
@Acb @RT(8)Action35 @F @T @RT(1)P @RT(0) @F @F @T @TL(6)
bReady := TRUE;
IF (sv_OperationMode <> nFullAutomatic) THEN
   sv_bAutoCycleRunning := FALSE;
END_IF;
g_SafetyData.MovementToActivate := 0;

@F

@Trans @RT(7)Trans15 @F @T @T @T @T @T @TL(2)
TRUE

@RT(7)Trans15 @F

@END_SfcData
@SaActions 6
@SaText @RT(11)ADelayCycle 1 @TL(17)
(**************************************** WARNING ********************************************
 *** The KEBA Kemro K2 System including software is not intended for safety control tasks! ***
 ***                       For further information see Comment tab!                        ***
 *********************************************************************************************)

//delay should not be executed in first cycle
IF sv_bFirstCycle THEN
   bDelayExceeded := TRUE;
ELSE
   IF sv_dCycleDelaySet > t#0s THEN
      sv_dCycleDelayAct := MIN(S_CheckStartCycle.T, sv_dCycleDelaySet);
   ELSE
      sv_dCycleDelayAct := t#0s;
   END_IF;
   bDelayExceeded := S_CheckStartCycle.T >= sv_dCycleDelaySet;
END_IF;

@SaText @RT(15)AEjectorAutoBwd 1 @TL(22)
(**************************************** WARNING ********************************************
 *** The KEBA Kemro K2 System including software is not intended for safety control tasks! ***
 ***                       For further information see Comment tab!                        ***
 *********************************************************************************************)

IF mbEjeBwdAtCycleStart AND NOT pbEjectorBwd^ AND NOT bEjectorBwdStarted THEN
   //only start ejector auto bwd movement if the ejector must be bwd at the beginning of the cycle
   //this information is taken from the safety array of the first step

   //modify pbActivated^ because otherwise the ejector will not move bwd if it is switched off
   sv_MovementsAvailable[iMoveNrEjectorBwd].pMovementData^.pbActivated := @sv_bTRUE;

   //attention:
   //if ejector is not programmed in sequence, there are no safety conditions for ejector bwd movement
   aStartSingleMovement(DeviceId := DeviceIdEjector,
                        MoveDir := cMoveBwd,
                        MoveId := cMoveBwd,
                        bNeedCheckSafety := sv_MovementsAvailable[iMoveNrEjectorBwd].pMovementData^.bProgrammedInSequence);

   bEjectorBwdStarted := TRUE;
END_IF;

@SaText @RT(15)AInitEjectorBwd 1 @TL(27)
(**************************************** WARNING ********************************************
 *** The KEBA Kemro K2 System including software is not intended for safety control tasks! ***
 ***                       For further information see Comment tab!                        ***
 *********************************************************************************************)

IF NOT bInitDone THEN
   fbGetMoveNumber(DeviceId := DeviceIdEjector,
                   MoveId := cMoveBwd,
                   MoveDir := cMoveBwd);

   IF fbGetMoveNumber.bFound THEN
      iMoveNrEjectorBwd := fbGetMoveNumber.iMoveNumber;
      pbEjectorBwd := sv_MovementsAvailable[fbGetMoveNumber.iMoveNumber].pMovementData^.pbPosReached;
      pbEjectorBwdActivated := sv_MovementsAvailable[fbGetMoveNumber.iMoveNumber].pMovementData^.pbActivated;
      pbEjectorReady := sv_MovementsAvailable[fbGetMoveNumber.iMoveNumber].pbDeviceReady;
   ELSE
      //ejector bwd movement not found
      pbEjectorBwd := @sv_bTRUE;
      pbEjectorBwdActivated := @sv_bTRUE;
      pbEjectorReady := @sv_bTRUE;
   END_IF;

   bInitDone := TRUE;
END_IF;

@SaText @RT(16)ACheckEjectorBwd 1 @TL(21)
(**************************************** WARNING ********************************************
 *** The KEBA Kemro K2 System including software is not intended for safety control tasks! ***
 ***                       For further information see Comment tab!                        ***
 *********************************************************************************************)

//set pbActivated to original reference
sv_MovementsAvailable[iMoveNrEjectorBwd].pMovementData^.pbActivated := pbEjectorBwdActivated;
bEjectorBwdStarted := FALSE;

IF NOT pbEjectorBwd^ THEN
   //ejector is not bwd -> set according alarm
   SET_ALARM(Name := sv_MovementsAvailable[iMoveNrEjectorBwd].pMovementData^.Alarm.AlarmId,
             SubID1 := sv_MovementsAvailable[iMoveNrEjectorBwd].pMovementData^.Alarm.SubId[1],
             SubID2 := sv_MovementsAvailable[iMoveNrEjectorBwd].pMovementData^.Alarm.SubId[2],
             SubID3 := sv_MovementsAvailable[iMoveNrEjectorBwd].pMovementData^.Alarm.SubId[3],
             SubID4 := sv_MovementsAvailable[iMoveNrEjectorBwd].pMovementData^.Alarm.SubId[4]);

   //switch to manual mode
   fbAutoManual();
END_IF;

@SaText @RT(16)AInitInterpreter 1 @TL(16)
(**************************************** WARNING ********************************************
 *** The KEBA Kemro K2 System including software is not intended for safety control tasks! ***
 ***                       For further information see Comment tab!                        ***
 *********************************************************************************************)

aClearStepState(TRUE);
abInterpreter.aInitInterpreter(iColumn := 1,
                               iRow := g_iAutoCycleLoopStartLine,
                               iEndRow := g_iAutoCycleLoopEndLine,
                               bSkipAlreadyPosReached := FALSE,
                               bExcludeActiveColumns := TRUE);

//find first "valid" line to save cycle time
abInterpreter.aIncreaseRow(iColumn := 1,
                           iEndRow := g_iAutoCycleLoopEndLine);

@SaText @RT(11)AStartCycle 1 @TL(24)
(**************************************** WARNING ********************************************
 *** The KEBA Kemro K2 System including software is not intended for safety control tasks! ***
 ***                       For further information see Comment tab!                        ***
 *********************************************************************************************)

IF NOT sv_bFirstCycle THEN
   //check of cycle time at the beginning of first cycle is not necessary
   aCheckCycleTime();
END_IF;

//save last cycle time
sv_dLastCycleTime := sv_dCycleTime;

mbCycleTimeRunning := TRUE;

//reset timers
mbResetCycleTime := TRUE;
mbResetCycleTimeMachine := TRUE;

sv_bAutoCycleRunning := TRUE;
mbCycleTimeMachineRunning := TRUE;

SET_EVENT(evNewCycleStarted);

@SaTrans 0
@SaExits 1
@SaExit @SaText @RT(12)StopAllMoves 1 @TL(2)
bStopCycle

@RT(8)stepname @RT(1)1 @T @F @SaSfc @RT(12)StopAllMoves 5 @RT(5)DUMMY
@BEG_SfcData 2
@ExitSeq @RT(4)sseq @F 3
@Step @RT(14)S_StopAllMoves @F @T @F @F @RT(0) @F
@AcbCont @RT(7)unnamed @F 1
@Acb @RT(16)AStopInterpreter @F @T @RT(1)P @RT(0) @F @F @T @TL(2)
abInterpreter.aStopInterpreterNormal();

@F

@Trans @RT(11)T_CheckStop @F @T @F @F @T @T @TL(2)
TRUE

@RT(7)Trans12 @F
@Goto @RT(16)S_CheckStartCond @F @F
@END_SfcData

@END_SfcBody

@@@BEG_Comment@@@
@TL(1)
Run the autocycle by calling the interpreter.
@@@END_Comment@@@

@BEG_Body
@TL(21)
(**************************************** WARNING ********************************************
 *** The KEBA Kemro K2 System including software is not intended for safety control tasks! ***
 ***                       For further information see Comment tab!                        ***
 *********************************************************************************************)

//call autoCycle
aRunAutoCycle(bStopCycle := mbStopCycle,
              bStopAfterCycle := mbStopAfterCycle);

IF aRunAutoCycle.bReady AND (mbStopCycle OR mbStopAfterCycle) THEN
   sv_bAutoCycleRunning := FALSE;
   // switch to manual mode and stop self at end of cycle
   fbAutoManual();

   abInterpreter.aResetStepMode();
   STOP_PROCESS_ALGORITHM(paCycleTime);
   STOP_PROCESS_ALGORITHM(paCycleTimeMachine);
   STOP_PROCESS_ALGORITHM();
END_IF;

@END_Body

@@@BEG_Comment@@@
@TL(3)
Run the auto cycle.
When the cycle has finished and mbStopCycle OR mbStopAfterCycle are true
opmode is automatically switched to manual and the PROCESS_ALGORITHM stops itself.
@@@END_Comment@@@

@BEG_Body
@TL(20)
(**************************************** WARNING ********************************************
 *** The KEBA Kemro K2 System including software is not intended for safety control tasks! ***
 ***                       For further information see Comment tab!                        ***
 *********************************************************************************************)

fbDebugTrace2(nODCInterpreter,'Reloading ODC files because of sv_bInitDone');

IF sv_bUseProgramSwitches THEN
   //use program switches
   aSetPendingRecalc(RecalcMode := nODCRecalcReloadFiles);
ELSE
   //use existing sequence and only recalc internal arrays
   aSetPendingRecalc(RecalcMode := nODCRecalcInternal);
END_IF;

aDoPendingRecalc();
IF aDoPendingRecalc.bStartedRecalc THEN
   fbDebugTrace2(nDeviceState, 'recalc because pInitDone');
END_IF;

@END_Body

@@@BEG_Comment@@@
@TL(1)
Cause initialisation of ODC sequence after startup(sv_bInitDone)
@@@END_Comment@@@

@BEG_Body
@TL(21)
(**************************************** WARNING ********************************************
 *** The KEBA Kemro K2 System including software is not intended for safety control tasks! ***
 ***                       For further information see Comment tab!                        ***
 *********************************************************************************************)

//initialize semaphore
Status := MovementsSema.Put();
IF Status <> KRTOS_Status_OK THEN
   dummy2 := ASSERT(FALSE, erAssert);
END_IF;

swoState := KSWO_AddVariable(Task := TaskInject,
                           Name := 'ActCycleTime',
                           Variable := sv_dCycleTime);

swoState := KSWO_AddVariable(Task := TaskAnalog,
                           Name := 'ActCycleTime',
                           Variable := sv_dCycleTime);

STOP_PROCESS_ALGORITHM();

@END_Body

@@@BEG_Comment@@@
@TL(0)

@@@END_Comment@@@

@BEG_Body
@TL(34)
(**************************************** WARNING ********************************************
 *** The KEBA Kemro K2 System including software is not intended for safety control tasks! ***
 ***                       For further information see Comment tab!                        ***
 *********************************************************************************************)

IF sv_OperationMode >= nHalfAutomatic THEN
   mbStopCycle := FALSE;
   mbStopAfterCycle := FALSE;
   (* back up sequence when machine is switched to auto mode
      and the sequence has changed *)
   START_PROCESS_ALGORITHM(paBackupSequence);

   (* PA stops itself again when finished *)
   START_PROCESS_ALGORITHM(paRunAutomaticMovements);
   START_PROCESS_ALGORITHM(paCycleTime);
   START_PROCESS_ALGORITHM(paCycleTimeMachine);
ELSIF sv_OperationMode < nHalfAutomatic THEN
   sv_bFirstCycle := TRUE;
   mbStopCycle := TRUE;
   mbCycleTimeRunning := FALSE;

   IF sv_StartedManualMovements.iStartedMovements = 0 THEN
      //recalc of sequence only if no movement is active
      //if there is still a movement active, the creation of a new sequence
      //will be triggered by postupdate algo pActiveMovements
      aDoPendingRecalc();
      IF aDoPendingRecalc.bStartedRecalc THEN
         fbDebugTrace2(nDeviceState, 'recalc because opmode change away from auto cycle');
      END_IF;
   END_IF;

END_IF;

@END_Body

@@@BEG_Comment@@@
@TL(3)
React to to operation mode changes and stop the autocycle immediately
when switching to setup/manual mode,
or reset cycle data when switching to Full/Halfauto operation mode.
@@@END_Comment@@@

@BEG_Body
@TL(7)
(**************************************** WARNING ********************************************
 *** The KEBA Kemro K2 System including software is not intended for safety control tasks! ***
 ***                       For further information see Comment tab!                        ***
 *********************************************************************************************)

mbStopAfterCycle := TRUE;

@END_Body

@@@BEG_Comment@@@
@TL(2)
Handle evAlarmFinishCycleAndStop event which signals to stop after the end
of the current autocycle
@@@END_Comment@@@

@BEG_Body
@TL(42)
(**************************************** WARNING ********************************************
 *** The KEBA Kemro K2 System including software is not intended for safety control tasks! ***
 ***                       For further information see Comment tab!                        ***
 *********************************************************************************************)
